LIN {X 0,Y 298.44,Z 121.432,A -85,B 0,C 180,E1 -16174.92,E2 -16174.92} C_VEL
LIN {X 0,Y 298.405,Z 121.429,A -85,B 0,C 180,E1 -16177.862,E2 -16177.862} C_VEL
LIN {X 0,Y 298.509,Z 121.421,A -85,B 0,C 180,E1 -16180.754,E2 -16180.754} C_VEL
LIN {X 0,Y 298.587,Z 121.413,A -85,B 0,C 180,E1 -16184.994,E2 -16184.994} C_VEL
LIN {X 0,Y 298.592,Z 121.415,A -85,B 0,C 180,E1 -16189.146,E2 -16189.146} C_VEL
LIN {X 0,Y 298.702,Z 121.391,A -85,B 0,C 180,E1 -16191.884,E2 -16191.884} C_VEL
LIN {X 0,Y 298.641,Z 121.406,A -85,B 0,C 180,E1 -16194.598,E2 -16194.598} C_VEL
LIN {X 0,Y 298.921,Z 121.375,A -85,B 0,C 180,E1 -16198.653,E2 -16198.653} C_VEL
LIN {X 0,Y 298.921,Z 121.361,A -85,B 0,C 180,E1 -16201.347,E2 -16201.347} C_VEL
LIN {X 0,Y 298.637,Z 121.402,A -85,B 0,C 180,E1 -16205.401,E2 -16205.401} C_VEL
LIN {X 0,Y 298.708,Z 121.401,A -85,B 0,C 180,E1 -16208.82,E2 -16208.82} C_VEL
LIN {X 0,Y 298.553,Z 121.423,A -85,B 0,C 180,E1 -16213.615,E2 -16213.615} C_VEL
LIN {X 0,Y 298.55,Z 121.407,A -85,B 0,C 180,E1 -16216.408,E2 -16216.408} C_VEL
LIN {X 0,Y 298.512,Z 121.418,A -85,B 0,C 180,E1 -16219.654,E2 -16219.654} C_VEL
LIN {X 0,Y 298.458,Z 121.428,A -85,B 0,C 180,E1 -16223.597,E2 -16223.597} C_VEL
LIN {X 0,Y 298.49,Z 121.425,A -85,B 0,C 180,E1 -16226.574,E2 -16226.574} C_VEL
LIN {X 0,Y 298.421,Z 121.432,A -85,B 0,C 180,E1 -16229.641,E2 -16229.641} C_VEL
LIN {X 0,Y 298.396,Z 121.435,A -85,B 0,C 180,E1 -16232.8,E2 -16232.8} C_VEL
LIN {X 0,Y 298.445,Z 121.436,A -85,B 0,C 180,E1 -16236.807,E2 -16236.807} C_VEL
LIN {X 0,Y 298.387,Z 121.428,A -85,B 0,C 180,E1 -16241.087,E2 -16241.087} C_VEL
LIN {X 0,Y 298.399,Z 121.435,A -85,B 0,C 180,E1 -16243.103,E2 -16243.103} C_VEL
LIN {X 0,Y 298.403,Z 121.44,A -85,B 0,C 180,E1 -16246.921,E2 -16246.921} C_VEL
LIN {X 0,Y 298.451,Z 121.59,A -85,B 0,C 180,E1 -16249.382,E2 -16249.382} C_VEL
LIN {X 0,Y 301.266,Z 131.505,A -85,B 0,C 180,E1 -16253.033,E2 -16253.033} C_VEL
LIN {X 0,Y 302.836,Z 137.275,A -85,B 0,C 180,E1 -16254.962,E2 -16254.962} C_VEL
LIN {X 0,Y 311.936,Z 155.274,A -85,B 0,C 180,E1 -16256.733,E2 -16256.733} C_VEL
LIN {X 0,Y 318.709,Z 170.292,A -85,B 0,C 180,E1 -16258.005,E2 -16258.005} C_VEL
LIN {X 0,Y 321.734,Z 187.115,A -85,B 0,C 180,E1 -16258.816,E2 -16258.816} C_VEL
LIN {X 0,Y 318.655,Z 274.997,A -85,B 0,C 180,E1 -16260.793,E2 -16260.793} C_VEL
LIN {X 0,Y 317.439,Z 289.664,A -85,B 0,C 180,E1 -16261.35,E2 -16261.35} C_VEL
LIN {X 0,Y 315.748,Z 303.63,A -85,B 0,C 180,E1 -16262.133,E2 -16262.133} C_VEL
LIN {X 0,Y 313.642,Z 317.483,A -85,B 0,C 180,E1 -16263.195,E2 -16263.195} C_VEL
LIN {X 0,Y 311.518,Z 330.032,A -85,B 0,C 180,E1 -16264.457,E2 -16264.457} C_VEL
LIN {X 0,Y 309.03,Z 342.414,A -85,B 0,C 180,E1 -16266.014,E2 -16266.014} C_VEL
LIN {X 0,Y 306.524,Z 353.602,A -85,B 0,C 180,E1 -16267.771,E2 -16267.771} C_VEL
LIN {X 0,Y 304.139,Z 363.638,A -85,B 0,C 180,E1 -16269.719,E2 -16269.719} C_VEL
LIN {X 0,Y 302.085,Z 371.989,A -85,B 0,C 180,E1 -16271.695,E2 -16271.695} C_VEL
LIN {X 0,Y 300.202,Z 379.986,A -85,B 0,C 180,E1 -16274.033,E2 -16274.033} C_VEL
LIN {X 0,Y 298.771,Z 386.446,A -85,B 0,C 180,E1 -16276.395,E2 -16276.395} C_VEL
LIN {X 0,Y 297.529,Z 392.192,A -85,B 0,C 180,E1 -16279.107,E2 -16279.107} C_VEL
LIN {X 0,Y 296.852,Z 396.392,A -85,B 0,C 180,E1 -16281.833,E2 -16281.833} C_VEL
LIN {X 0,Y 296.531,Z 399.17,A -85,B 0,C 180,E1 -16284.56,E2 -16284.56} C_VEL
LIN {X 0,Y 296.512,Z 400.597,A -85,B 0,C 180,E1 -16287.283,E2 -16287.283} C_VEL
LIN {X 0,Y 296.479,Z 400.691,A -85,B 0,C 180,E1 -16290,E2 -16290} C_VEL
LIN {X 0,Y 296.518,Z 399.447,A -85,B 0,C 180,E1 -16292.717,E2 -16292.717} C_VEL
LIN {X 0,Y 296.511,Z 396.814,A -85,B 0,C 180,E1 -16295.44,E2 -16295.44} C_VEL
LIN {X 0,Y 296.783,Z 392.722,A -85,B 0,C 180,E1 -16298.168,E2 -16298.168} C_VEL
LIN {X 0,Y 297.314,Z 387.046,A -85,B 0,C 180,E1 -16300.9,E2 -16300.9} C_VEL
LIN {X 0,Y 298.285,Z 380.643,A -85,B 0,C 180,E1 -16303.281,E2 -16303.281} C_VEL
LIN {X 0,Y 299.321,Z 373.124,A -85,B 0,C 180,E1 -16305.534,E2 -16305.534} C_VEL
LIN {X 0,Y 300.776,Z 364.3,A -85,B 0,C 180,E1 -16307.683,E2 -16307.683} C_VEL
LIN {X 0,Y 302.455,Z 354.225,A -85,B 0,C 180,E1 -16309.69,E2 -16309.69} C_VEL
LIN {X 0,Y 304.398,Z 343.006,A -85,B 0,C 180,E1 -16311.501,E2 -16311.501} C_VEL
LIN {X 0,Y 306.181,Z 331.827,A -85,B 0,C 180,E1 -16312.968,E2 -16312.968} C_VEL
LIN {X 0,Y 307.925,Z 319.653,A -85,B 0,C 180,E1 -16314.256,E2 -16314.256} C_VEL
LIN {X 0,Y 309.491,Z 306.12,A -85,B 0,C 180,E1 -16315.38,E2 -16315.38} C_VEL
LIN {X 0,Y 310.912,Z 291.992,A -85,B 0,C 180,E1 -16316.244,E2 -16316.244} C_VEL
LIN {X 0,Y 311.897,Z 278.189,A -85,B 0,C 180,E1 -16316.831,E2 -16316.831} C_VEL
LIN {X 0,Y 312.684,Z 257.755,A -85,B 0,C 180,E1 -16317.346,E2 -16317.346} C_VEL
LIN {X 0,Y 314.615,Z 183.423,A -85,B 0,C 180,E1 -16319.027,E2 -16319.027} C_VEL
LIN {X 0,Y 310.494,Z 157.724,A -85,B 0,C 180,E1 -16320.059,E2 -16320.059} C_VEL
LIN {X 0,Y 302.188,Z 137.332,A -85,B 0,C 180,E1 -16321.449,E2 -16321.449} C_VEL
LIN {X 0,Y 299.625,Z 126.323,A -85,B 0,C 180,E1 -16324.819,E2 -16324.819} C_VEL
LIN {X 0,Y 298.467,Z 121.436,A -85,B 0,C 180,E1 -16326.436,E2 -16326.436} C_VEL
LIN {X 0,Y 298.408,Z 121.44,A -85,B 0,C 180,E1 -16329.486,E2 -16329.486} C_VEL
LIN {X 0,Y 298.425,Z 121.436,A -85,B 0,C 180,E1 -16333.109,E2 -16333.109} C_VEL
LIN {X 0,Y 298.466,Z 121.429,A -85,B 0,C 180,E1 -16336.932,E2 -16336.932} C_VEL
LIN {X 0,Y 298.428,Z 121.425,A -85,B 0,C 180,E1 -16341,E2 -16341} C_VEL
LIN {X 0,Y 298.43,Z 121.436,A -85,B 0,C 180,E1 -16343.932,E2 -16343.932} C_VEL
LIN {X 0,Y 298.394,Z 121.439,A -85,B 0,C 180,E1 -16347.983,E2 -16347.983} C_VEL
LIN {X 0,Y 298.468,Z 121.429,A -85,B 0,C 180,E1 -16351.905,E2 -16351.905} C_VEL
LIN {X 0,Y 298.485,Z 121.428,A -85,B 0,C 180,E1 -16354.924,E2 -16354.924} C_VEL
LIN {X 0,Y 298.449,Z 121.432,A -85,B 0,C 180,E1 -16359.315,E2 -16359.315} C_VEL
LIN {X 0,Y 298.537,Z 121.417,A -85,B 0,C 180,E1 -16362.179,E2 -16362.179} C_VEL
LIN {X 0,Y 298.592,Z 121.416,A -85,B 0,C 180,E1 -16364.995,E2 -16364.995} C_VEL
LIN {X 0,Y 298.592,Z 121.414,A -85,B 0,C 180,E1 -16369.147,E2 -16369.147} C_VEL
LIN {X 0,Y 298.744,Z 121.395,A -85,B 0,C 180,E1 -16371.886,E2 -16371.886} C_VEL
LIN {X 0,Y 298.655,Z 121.403,A -85,B 0,C 180,E1 -16374.599,E2 -16374.599} C_VEL
LIN {X 0,Y 298.921,Z 121.374,A -85,B 0,C 180,E1 -16378.653,E2 -16378.653} C_VEL
LIN {X 0,Y 298.921,Z 121.366,A -85,B 0,C 180,E1 -16381.347,E2 -16381.347} C_VEL
LIN {X 0,Y 298.644,Z 121.407,A -85,B 0,C 180,E1 -16385.402,E2 -16385.402} C_VEL
LIN {X 0,Y 298.712,Z 121.398,A -85,B 0,C 180,E1 -16388.116,E2 -16388.116} C_VEL
LIN {X 0,Y 298.553,Z 121.42,A -85,B 0,C 180,E1 -16392.232,E2 -16392.232} C_VEL
LIN {X 0,Y 298.605,Z 121.412,A -85,B 0,C 180,E1 -16395.209,E2 -16395.209} C_VEL
LIN {X 0,Y 298.539,Z 121.417,A -85,B 0,C 180,E1 -16399.243,E2 -16399.243} C_VEL
LIN {X 0,Y 298.457,Z 121.429,A -85,B 0,C 180,E1 -16403.598,E2 -16403.598} C_VEL
LIN {X 0,Y 298.486,Z 121.424,A -85,B 0,C 180,E1 -16406.575,E2 -16406.575} C_VEL
LIN {X 0,Y 298.416,Z 121.436,A -85,B 0,C 180,E1 -16409.642,E2 -16409.642} C_VEL
LIN {X 0,Y 298.395,Z 121.436,A -85,B 0,C 180,E1 -16412.801,E2 -16412.801} C_VEL
LIN {X 0,Y 298.444,Z 121.431,A -85,B 0,C 180,E1 -16416.807,E2 -16416.807} C_VEL
LIN {X 0,Y 298.388,Z 121.439,A -85,B 0,C 180,E1 -16421.088,E2 -16421.088} C_VEL
LIN {X 0,Y 298.389,Z 121.439,A -85,B 0,C 180,E1 -16425.042,E2 -16425.042} C_VEL
LIN {X 0,Y 298.388,Z 121.439,A -85,B 0,C 180,E1 -16428.913,E2 -16428.913} C_VEL
LIN {X 0,Y 298.445,Z 121.435,A -85,B 0,C 180,E1 -16433.194,E2 -16433.194} C_VEL
LIN {X 0,Y 298.394,Z 121.44,A -85,B 0,C 180,E1 -16437.2,E2 -16437.2} C_VEL
LIN {X 0,Y 298.404,Z 121.44,A -85,B 0,C 180,E1 -16440.625,E2 -16440.625} C_VEL
LIN {X 0,Y 298.436,Z 121.472,A -85,B 0,C 180,E1 -16442.873,E2 -16442.873} C_VEL
LIN {X 0,Y 299.591,Z 126.094,A -85,B 0,C 180,E1 -16444.382,E2 -16444.382} C_VEL
LIN {X 0,Y 308.871,Z 146.99,A -85,B 0,C 180,E1 -16445.883,E2 -16445.883} C_VEL
LIN {X 0,Y 314.918,Z 162.698,A -85,B 0,C 180,E1 -16446.857,E2 -16446.857} C_VEL
LIN {X 0,Y 315.167,Z 165.643,A -85,B 0,C 180,E1 -16446.953,E2 -16446.953} C_VEL
LIN {X 0,Y 312.39,Z 262.581,A -85,B 0,C 180,E1 -16449.161,E2 -16449.161} C_VEL
LIN {X 0,Y 311.659,Z 276.3,A -85,B 0,C 180,E1 -16449.714,E2 -16449.714} C_VEL
LIN {X 0,Y 310.527,Z 289.807,A -85,B 0,C 180,E1 -16450.499,E2 -16450.499} C_VEL
LIN {X 0,Y 309.152,Z 302.098,A -85,B 0,C 180,E1 -16451.442,E2 -16451.442} C_VEL
LIN {X 0,Y 307.636,Z 313.548,A -85,B 0,C 180,E1 -16452.552,E2 -16452.552} C_VEL
LIN {X 0,Y 305.934,Z 325.457,A -85,B 0,C 180,E1 -16453.998,E2 -16453.998} C_VEL
LIN {X 0,Y 304.144,Z 336.336,A -85,B 0,C 180,E1 -16455.617,E2 -16455.617} C_VEL
LIN {X 0,Y 302.338,Z 346.911,A -85,B 0,C 180,E1 -16457.55,E2 -16457.55} C_VEL
LIN {X 0,Y 300.8,Z 355.936,A -85,B 0,C 180,E1 -16459.568,E2 -16459.568} C_VEL
LIN {X 0,Y 299.495,Z 363.328,A -85,B 0,C 180,E1 -16461.567,E2 -16461.567} C_VEL
LIN {X 0,Y 298.331,Z 370.395,A -85,B 0,C 180,E1 -16463.915,E2 -16463.915} C_VEL
LIN {X 0,Y 297.515,Z 375.339,A -85,B 0,C 180,E1 -16465.936,E2 -16465.936} C_VEL
LIN {X 0,Y 296.911,Z 380.438,A -85,B 0,C 180,E1 -16468.644,E2 -16468.644} C_VEL
LIN {X 0,Y 296.563,Z 384.053,A -85,B 0,C 180,E1 -16471.358,E2 -16471.358} C_VEL
LIN {X 0,Y 296.519,Z 386.28,A -85,B 0,C 180,E1 -16474.078,E2 -16474.078} C_VEL
LIN {X 0,Y 296.502,Z 387.182,A -85,B 0,C 180,E1 -16476.807,E2 -16476.807} C_VEL
LIN {X 0,Y 296.471,Z 386.764,A -85,B 0,C 180,E1 -16479.552,E2 -16479.552} C_VEL
LIN {X 0,Y 296.862,Z 385.003,A -85,B 0,C 180,E1 -16482.302,E2 -16482.302} C_VEL
LIN {X 0,Y 297.563,Z 381.854,A -85,B 0,C 180,E1 -16485.059,E2 -16485.059} C_VEL
LIN {X 0,Y 298.555,Z 377.171,A -85,B 0,C 180,E1 -16487.82,E2 -16487.82} C_VEL
LIN {X 0,Y 300.087,Z 371.034,A -85,B 0,C 180,E1 -16490.479,E2 -16490.479} C_VEL
LIN {X 0,Y 301.9,Z 363.692,A -85,B 0,C 180,E1 -16492.95,E2 -16492.95} C_VEL
LIN {X 0,Y 304.088,Z 355.073,A -85,B 0,C 180,E1 -16495.254,E2 -16495.254} C_VEL
LIN {X 0,Y 306.353,Z 345.552,A -85,B 0,C 180,E1 -16497.311,E2 -16497.311} C_VEL
LIN {X 0,Y 308.651,Z 335.233,A -85,B 0,C 180,E1 -16499.125,E2 -16499.125} C_VEL
LIN {X 0,Y 311.156,Z 323.794,A -85,B 0,C 180,E1 -16500.736,E2 -16500.736} C_VEL
LIN {X 0,Y 313.123,Z 312.72,A -85,B 0,C 180,E1 -16502.023,E2 -16502.023} C_VEL
LIN {X 0,Y 315.343,Z 299.818,A -85,B 0,C 180,E1 -16503.19,E2 -16503.19} C_VEL
LIN {X 0,Y 316.836,Z 287.775,A -85,B 0,C 180,E1 -16504.062,E2 -16504.062} C_VEL
LIN {X 0,Y 318.183,Z 273.727,A -85,B 0,C 180,E1 -16504.809,E2 -16504.809} C_VEL
LIN {X 0,Y 319.144,Z 259.623,A -85,B 0,C 180,E1 -16505.297,E2 -16505.297} C_VEL
LIN {X 0,Y 322.223,Z 171.012,A -85,B 0,C 180,E1 -16507.278,E2 -16507.278} C_VEL
LIN {X 0,Y 314.561,Z 154.009,A -85,B 0,C 180,E1 -16508.687,E2 -16508.687} C_VEL
LIN {X 0,Y 308.153,Z 141.521,A -85,B 0,C 180,E1 -16509.891,E2 -16509.891} C_VEL
LIN {X 0,Y 305.295,Z 136.304,A -85,B 0,C 180,E1 -16510.441,E2 -16510.441} C_VEL
LIN {X 0,Y 303.417,Z 133.303,A -85,B 0,C 180,E1 -16510.813,E2 -16510.813} C_VEL
LIN {X 0,Y 300.871,Z 131.097,A -85,B 0,C 180,E1 -16511.261,E2 -16511.261} C_VEL
LIN {X 0,Y 292.931,Z 126.669,A -85,B 0,C 180,E1 -16512.655,E2 -16512.655} C_VEL
LIN {X 0,Y 292.253,Z 125.838,A -85,B 0,C 180,E1 -16512.971,E2 -16512.971} C_VEL
LIN {X 0,Y 291.325,Z 122.315,A -85,B 0,C 180,E1 -16514.471,E2 -16514.471} C_VEL
LIN {X 0,Y 291.296,Z 122.321,A -85,B 0,C 180,E1 -16518.411,E2 -16518.411} C_VEL
LIN {X 0,Y 291.387,Z 122.315,A -85,B 0,C 180,E1 -16522.916,E2 -16522.916} C_VEL
LIN {X 0,Y 291.345,Z 122.316,A -85,B 0,C 180,E1 -16526.301,E2 -16526.301} C_VEL
LIN {X 0,Y 291.366,Z 122.308,A -85,B 0,C 180,E1 -16530.268,E2 -16530.268} C_VEL
LIN {X 0,Y 291.36,Z 122.309,A -85,B 0,C 180,E1 -16534.266,E2 -16534.266} C_VEL
LIN {X 0,Y 291.366,Z 122.306,A -85,B 0,C 180,E1 -16537.298,E2 -16537.298} C_VEL
LIN {X 0,Y 291.46,Z 122.305,A -85,B 0,C 180,E1 -16540.27,E2 -16540.27} C_VEL
LIN {X 0,Y 291.499,Z 122.298,A -85,B 0,C 180,E1 -16544.665,E2 -16544.665} C_VEL
LIN {X 0,Y 291.536,Z 122.295,A -85,B 0,C 180,E1 -16548.88,E2 -16548.88} C_VEL
LIN {X 0,Y 291.655,Z 122.267,A -85,B 0,C 180,E1 -16551.687,E2 -16551.687} C_VEL
LIN {X 0,Y 291.61,Z 122.283,A -85,B 0,C 180,E1 -16554.468,E2 -16554.468} C_VEL
LIN {X 0,Y 291.887,Z 122.251,A -85,B 0,C 180,E1 -16558.62,E2 -16558.62} C_VEL
LIN {X 0,Y 291.887,Z 122.237,A -85,B 0,C 180,E1 -16561.379,E2 -16561.379} C_VEL
LIN {X 0,Y 291.606,Z 122.276,A -85,B 0,C 180,E1 -16565.532,E2 -16565.532} C_VEL
LIN {X 0,Y 291.668,Z 122.278,A -85,B 0,C 180,E1 -16568.91,E2 -16568.91} C_VEL
LIN {X 0,Y 291.519,Z 122.291,A -85,B 0,C 180,E1 -16572.531,E2 -16572.531} C_VEL
LIN {X 0,Y 291.556,Z 122.282,A -85,B 0,C 180,E1 -16575.376,E2 -16575.376} C_VEL
LIN {X 0,Y 291.452,Z 122.297,A -85,B 0,C 180,E1 -16579.875,E2 -16579.875} C_VEL
LIN {X 0,Y 291.401,Z 122.304,A -85,B 0,C 180,E1 -16584.205,E2 -16584.205} C_VEL
LIN {X 0,Y 291.423,Z 122.307,A -85,B 0,C 180,E1 -16587.271,E2 -16587.271} C_VEL
LIN {X 0,Y 291.338,Z 122.318,A -85,B 0,C 180,E1 -16590.437,E2 -16590.437} C_VEL
LIN {X 0,Y 291.345,Z 122.319,A -85,B 0,C 180,E1 -16593.698,E2 -16593.698} C_VEL
LIN {X 0,Y 291.373,Z 122.316,A -85,B 0,C 180,E1 -16597.253,E2 -16597.253} C_VEL
LIN {X 0,Y 291.332,Z 122.3,A -85,B 0,C 180,E1 -16600.642,E2 -16600.642} C_VEL
LIN {X 0,Y 291.29,Z 122.308,A -85,B 0,C 180,E1 -16604.402,E2 -16604.402} C_VEL
LIN {X 0,Y 291.367,Z 122.352,A -85,B 0,C 180,E1 -16608.395,E2 -16608.395} C_VEL
LIN {X 0,Y 294.066,Z 131.907,A -85,B 0,C 180,E1 -16612.062,E2 -16612.062} C_VEL
LIN {X 0,Y 295.437,Z 136.791,A -85,B 0,C 180,E1 -16613.836,E2 -16613.836} C_VEL
LIN {X 0,Y 303.07,Z 151.502,A -85,B 0,C 180,E1 -16615.411,E2 -16615.411} C_VEL
LIN {X 0,Y 311.133,Z 168.352,A -85,B 0,C 180,E1 -16616.991,E2 -16616.991} C_VEL
LIN {X 0,Y 313.243,Z 173.632,A -85,B 0,C 180,E1 -16617.41,E2 -16617.41} C_VEL
LIN {X 0,Y 315.791,Z 188.416,A -85,B 0,C 180,E1 -16618.133,E2 -16618.133} C_VEL
LIN {X 0,Y 312.601,Z 275.339,A -85,B 0,C 180,E1 -16620.124,E2 -16620.124} C_VEL
LIN {X 0,Y 311.345,Z 289.824,A -85,B 0,C 180,E1 -16620.689,E2 -16620.689} C_VEL
LIN {X 0,Y 309.516,Z 304.269,A -85,B 0,C 180,E1 -16621.521,E2 -16621.521} C_VEL
LIN {X 0,Y 307.347,Z 317.946,A -85,B 0,C 180,E1 -16622.6,E2 -16622.6} C_VEL
LIN {X 0,Y 305.174,Z 330.231,A -85,B 0,C 180,E1 -16623.868,E2 -16623.868} C_VEL
LIN {X 0,Y 302.569,Z 342.657,A -85,B 0,C 180,E1 -16625.468,E2 -16625.468} C_VEL
LIN {X 0,Y 299.964,Z 353.753,A -85,B 0,C 180,E1 -16627.258,E2 -16627.258} C_VEL
LIN {X 0,Y 297.459,Z 363.736,A -85,B 0,C 180,E1 -16629.243,E2 -16629.243} C_VEL
LIN {X 0,Y 295.002,Z 373.271,A -85,B 0,C 180,E1 -16631.599,E2 -16631.599} C_VEL
LIN {X 0,Y 293.363,Z 379.811,A -85,B 0,C 180,E1 -16633.584,E2 -16633.584} C_VEL
LIN {X 0,Y 291.848,Z 386.424,A -85,B 0,C 180,E1 -16636.065,E2 -16636.065} C_VEL
LIN {X 0,Y 290.524,Z 392.137,A -85,B 0,C 180,E1 -16638.841,E2 -16638.841} C_VEL
LIN {X 0,Y 289.809,Z 396.306,A -85,B 0,C 180,E1 -16641.633,E2 -16641.633} C_VEL
LIN {X 0,Y 289.426,Z 399.204,A -85,B 0,C 180,E1 -16644.614,E2 -16644.614} C_VEL
LIN {X 0,Y 289.416,Z 400.454,A -85,B 0,C 180,E1 -16647.216,E2 -16647.216} C_VEL
LIN {X 0,Y 289.398,Z 400.52,A -85,B 0,C 180,E1 -16650,E2 -16650} C_VEL
LIN {X 0,Y 289.421,Z 399.241,A -85,B 0,C 180,E1 -16652.783,E2 -16652.783} C_VEL
LIN {X 0,Y 289.434,Z 396.574,A -85,B 0,C 180,E1 -16655.574,E2 -16655.574} C_VEL
LIN {X 0,Y 289.718,Z 392.45,A -85,B 0,C 180,E1 -16658.369,E2 -16658.369} C_VEL
LIN {X 0,Y 290.122,Z 388.36,A -85,B 0,C 180,E1 -16660.467,E2 -16660.467} C_VEL
LIN {X 0,Y 290.841,Z 383.247,A -85,B 0,C 180,E1 -16662.561,E2 -16662.561} C_VEL
LIN {X 0,Y 292.008,Z 375.941,A -85,B 0,C 180,E1 -16664.994,E2 -16664.994} C_VEL
LIN {X 0,Y 293.136,Z 368.263,A -85,B 0,C 180,E1 -16667.079,E2 -16667.079} C_VEL
LIN {X 0,Y 294.815,Z 359.054,A -85,B 0,C 180,E1 -16669.134,E2 -16669.134} C_VEL
LIN {X 0,Y 296.386,Z 349.857,A -85,B 0,C 180,E1 -16670.835,E2 -16670.835} C_VEL
LIN {X 0,Y 298.382,Z 338.889,A -85,B 0,C 180,E1 -16672.504,E2 -16672.504} C_VEL
LIN {X 0,Y 300.217,Z 326.747,A -85,B 0,C 180,E1 -16674.013,E2 -16674.013} C_VEL
LIN {X 0,Y 301.87,Z 315.299,A -85,B 0,C 180,E1 -16675.143,E2 -16675.143} C_VEL
LIN {X 0,Y 303.311,Z 302.88,A -85,B 0,C 180,E1 -16676.119,E2 -16676.119} C_VEL
LIN {X 0,Y 304.703,Z 288.433,A -85,B 0,C 180,E1 -16676.96,E2 -16676.96} C_VEL
LIN {X 0,Y 305.701,Z 273.863,A -85,B 0,C 180,E1 -16677.513,E2 -16677.513} C_VEL
LIN {X 0,Y 308.253,Z 184.312,A -85,B 0,C 180,E1 -16679.592,E2 -16679.592} C_VEL
LIN {X 0,Y 304.502,Z 160.641,A -85,B 0,C 180,E1 -16680.568,E2 -16680.568} C_VEL
LIN {X 0,Y 297.951,Z 144.295,A -85,B 0,C 180,E1 -16681.677,E2 -16681.677} C_VEL
LIN {X 0,Y 294.952,Z 137.255,A -85,B 0,C 180,E1 -16682.196,E2 -16682.196} C_VEL
LIN {X 0,Y 292.386,Z 126.362,A -85,B 0,C 180,E1 -16685.653,E2 -16685.653} C_VEL
LIN {X 0,Y 291.428,Z 122.313,A -85,B 0,C 180,E1 -16687.023,E2 -16687.023} C_VEL
LIN {X 0,Y 291.334,Z 122.319,A -85,B 0,C 180,E1 -16690.642,E2 -16690.642} C_VEL
LIN {X 0,Y 291.341,Z 122.318,A -85,B 0,C 180,E1 -16694.392,E2 -16694.392} C_VEL
LIN {X 0,Y 291.386,Z 122.312,A -85,B 0,C 180,E1 -16698.391,E2 -16698.391} C_VEL
LIN {X 0,Y 291.376,Z 122.301,A -85,B 0,C 180,E1 -16701.162,E2 -16701.162} C_VEL
LIN {X 0,Y 291.384,Z 122.312,A -85,B 0,C 180,E1 -16704.629,E2 -16704.629} C_VEL
LIN {X 0,Y 291.371,Z 122.315,A -85,B 0,C 180,E1 -16707.951,E2 -16707.951} C_VEL
LIN {X 0,Y 291.384,Z 122.311,A -85,B 0,C 180,E1 -16711.159,E2 -16711.159} C_VEL
LIN {X 0,Y 291.419,Z 122.307,A -85,B 0,C 180,E1 -16714.272,E2 -16714.272} C_VEL
LIN {X 0,Y 291.38,Z 122.315,A -85,B 0,C 180,E1 -16717.3,E2 -16717.3} C_VEL
LIN {X 0,Y 291.457,Z 122.301,A -85,B 0,C 180,E1 -16720.27,E2 -16720.27} C_VEL
LIN {X 0,Y 291.554,Z 122.294,A -85,B 0,C 180,E1 -16724.624,E2 -16724.624} C_VEL
LIN {X 0,Y 291.535,Z 122.293,A -85,B 0,C 180,E1 -16728.881,E2 -16728.881} C_VEL
LIN {X 0,Y 291.696,Z 122.273,A -85,B 0,C 180,E1 -16731.688,E2 -16731.688} C_VEL
LIN {X 0,Y 291.626,Z 122.277,A -85,B 0,C 180,E1 -16734.468,E2 -16734.468} C_VEL
LIN {X 0,Y 291.887,Z 122.251,A -85,B 0,C 180,E1 -16738.621,E2 -16738.621} C_VEL
LIN {X 0,Y 291.887,Z 122.241,A -85,B 0,C 180,E1 -16741.38,E2 -16741.38} C_VEL
LIN {X 0,Y 291.659,Z 122.275,A -85,B 0,C 180,E1 -16746.552,E2 -16746.552} C_VEL
LIN {X 0,Y 291.571,Z 122.282,A -85,B 0,C 180,E1 -16749.714,E2 -16749.714} C_VEL
LIN {X 0,Y 291.521,Z 122.298,A -85,B 0,C 180,E1 -16753.951,E2 -16753.951} C_VEL
LIN {X 0,Y 291.486,Z 122.293,A -85,B 0,C 180,E1 -16756.818,E2 -16756.818} C_VEL
LIN {X 0,Y 291.45,Z 122.305,A -85,B 0,C 180,E1 -16759.875,E2 -16759.875} C_VEL
LIN {X 0,Y 291.4,Z 122.303,A -85,B 0,C 180,E1 -16764.206,E2 -16764.206} C_VEL
LIN {X 0,Y 291.42,Z 122.308,A -85,B 0,C 180,E1 -16767.272,E2 -16767.272} C_VEL
LIN {X 0,Y 291.334,Z 122.315,A -85,B 0,C 180,E1 -16770.438,E2 -16770.438} C_VEL
LIN {X 0,Y 291.344,Z 122.318,A -85,B 0,C 180,E1 -16773.699,E2 -16773.699} C_VEL
LIN {X 0,Y 291.372,Z 122.311,A -85,B 0,C 180,E1 -16777.253,E2 -16777.253} C_VEL
LIN {X 0,Y 291.333,Z 122.321,A -85,B 0,C 180,E1 -16780.643,E2 -16780.643} C_VEL
LIN {X 0,Y 291.315,Z 122.323,A -85,B 0,C 180,E1 -16784.398,E2 -16784.398} C_VEL
LIN {X 0,Y 291.328,Z 122.322,A -85,B 0,C 180,E1 -16788.405,E2 -16788.405} C_VEL
LIN {X 0,Y 291.348,Z 122.305,A -85,B 0,C 180,E1 -16791.158,E2 -16791.158} C_VEL
LIN {X 0,Y 291.362,Z 122.318,A -85,B 0,C 180,E1 -16794.627,E2 -16794.627} C_VEL
LIN {X 0,Y 291.367,Z 122.316,A -85,B 0,C 180,E1 -16797.95,E2 -16797.95} C_VEL
LIN {X 0,Y 291.39,Z 122.313,A -85,B 0,C 180,E1 -16802.141,E2 -16802.141} C_VEL
LIN {X 0,Y 291.397,Z 122.542,A -85,B 0,C 180,E1 -16802.337,E2 -16802.337} C_VEL
LIN {X 0,Y 292.364,Z 126.299,A -85,B 0,C 180,E1 -16803.591,E2 -16803.591} C_VEL
LIN {X 0,Y 300.522,Z 144.106,A -85,B 0,C 180,E1 -16804.964,E2 -16804.964} C_VEL
LIN {X 0,Y 307.832,Z 162.323,A -85,B 0,C 180,E1 -16806.178,E2 -16806.178} C_VEL
LIN {X 0,Y 308.799,Z 165.052,A -85,B 0,C 180,E1 -16806.341,E2 -16806.341} C_VEL
LIN {X 0,Y 305.952,Z 262.733,A -85,B 0,C 180,E1 -16808.613,E2 -16808.613} C_VEL
LIN {X 0,Y 305.187,Z 276.458,A -85,B 0,C 180,E1 -16809.176,E2 -16809.176} C_VEL
LIN {X 0,Y 304.024,Z 289.966,A -85,B 0,C 180,E1 -16809.976,E2 -16809.976} C_VEL
LIN {X 0,Y 302.483,Z 303.136,A -85,B 0,C 180,E1 -16811.018,E2 -16811.018} C_VEL
LIN {X 0,Y 300.93,Z 314.417,A -85,B 0,C 180,E1 -16812.15,E2 -16812.15} C_VEL
LIN {X 0,Y 299.145,Z 326.205,A -85,B 0,C 180,E1 -16813.625,E2 -16813.625} C_VEL
LIN {X 0,Y 297.312,Z 336.984,A -85,B 0,C 180,E1 -16815.279,E2 -16815.279} C_VEL
LIN {X 0,Y 295.509,Z 347.152,A -85,B 0,C 180,E1 -16817.187,E2 -16817.187} C_VEL
LIN {X 0,Y 293.859,Z 356.435,A -85,B 0,C 180,E1 -16819.319,E2 -16819.319} C_VEL
LIN {X 0,Y 292.497,Z 363.769,A -85,B 0,C 180,E1 -16821.363,E2 -16821.363} C_VEL
LIN {X 0,Y 291.279,Z 370.784,A -85,B 0,C 180,E1 -16823.767,E2 -16823.767} C_VEL
LIN {X 0,Y 290.443,Z 375.68,A -85,B 0,C 180,E1 -16825.837,E2 -16825.837} C_VEL
LIN {X 0,Y 290.013,Z 379.632,A -85,B 0,C 180,E1 -16827.917,E2 -16827.917} C_VEL
LIN {X 0,Y 289.6,Z 382.699,A -85,B 0,C 180,E1 -16830,E2 -16830} C_VEL
LIN {X 0,Y 289.481,Z 385.567,A -85,B 0,C 180,E1 -16832.783,E2 -16832.783} C_VEL
LIN {X 0,Y 289.434,Z 387.089,A -85,B 0,C 180,E1 -16835.574,E2 -16835.574} C_VEL
LIN {X 0,Y 289.337,Z 387.294,A -85,B 0,C 180,E1 -16838.38,E2 -16838.38} C_VEL
LIN {X 0,Y 289.528,Z 386.167,A -85,B 0,C 180,E1 -16841.198,E2 -16841.198} C_VEL
LIN {X 0,Y 290.183,Z 383.678,A -85,B 0,C 180,E1 -16844.016,E2 -16844.016} C_VEL
LIN {X 0,Y 291.051,Z 379.723,A -85,B 0,C 180,E1 -16846.844,E2 -16846.844} C_VEL
LIN {X 0,Y 292.469,Z 374.17,A -85,B 0,C 180,E1 -16849.659,E2 -16849.659} C_VEL
LIN {X 0,Y 294.109,Z 367.864,A -85,B 0,C 180,E1 -16852.109,E2 -16852.109} C_VEL
LIN {X 0,Y 296.215,Z 359.98,A -85,B 0,C 180,E1 -16854.532,E2 -16854.532} C_VEL
LIN {X 0,Y 298.363,Z 351.709,A -85,B 0,C 180,E1 -16856.587,E2 -16856.587} C_VEL
LIN {X 0,Y 300.755,Z 341.702,A -85,B 0,C 180,E1 -16858.623,E2 -16858.623} C_VEL
LIN {X 0,Y 303.124,Z 331.626,A -85,B 0,C 180,E1 -16860.284,E2 -16860.284} C_VEL
LIN {X 0,Y 305.711,Z 319.404,A -85,B 0,C 180,E1 -16861.921,E2 -16861.921} C_VEL
LIN {X 0,Y 307.97,Z 307.274,A -85,B 0,C 180,E1 -16863.209,E2 -16863.209} C_VEL
LIN {X 0,Y 309.989,Z 293.778,A -85,B 0,C 180,E1 -16864.33,E2 -16864.33} C_VEL
LIN {X 0,Y 311.6,Z 279.631,A -85,B 0,C 180,E1 -16865.209,E2 -16865.209} C_VEL
LIN {X 0,Y 312.793,Z 265.42,A -85,B 0,C 180,E1 -16865.812,E2 -16865.812} C_VEL
LIN {X 0,Y 313.742,Z 243.274,A -85,B 0,C 180,E1 -16866.369,E2 -16866.369} C_VEL
LIN {X 0,Y 316.316,Z 173.613,A -85,B 0,C 180,E1 -16867.93,E2 -16867.93} C_VEL
LIN {X 0,Y 310.974,Z 161.025,A -85,B 0,C 180,E1 -16868.961,E2 -16868.961} C_VEL
LIN {X 0,Y 303.586,Z 146.257,A -85,B 0,C 180,E1 -16870.396,E2 -16870.396} C_VEL
LIN {X 0,Y 296.791,Z 134.136,A -85,B 0,C 180,E1 -16871.761,E2 -16871.761} C_VEL
LIN {X 0,Y 292.475,Z 126.533,A -85,B 0,C 180,E1 -16872.686,E2 -16872.686} C_VEL
LIN {X 0,Y 292.253,Z 125.838,A -85,B 0,C 180,E1 -16872.971,E2 -16872.971} C_VEL
LIN {X 0,Y 291.13,Z 124.464,A -85,B 0,C 180,E1 -16873.674,E2 -16873.674} C_VEL
LIN {X 0,Y 287.887,Z 123.379,A -85,B 0,C 180,E1 -16874.828,E2 -16874.828} C_VEL
LIN {X 0,Y 284.903,Z 123.179,A -85,B 0,C 180,E1 -16876.049,E2 -16876.049} C_VEL
LIN {X 0,Y 284.209,Z 123.196,A -85,B 0,C 180,E1 -16876.847,E2 -16876.847} C_VEL
LIN {X 0,Y 284.257,Z 123.18,A -85,B 0,C 180,E1 -16880.036,E2 -16880.036} C_VEL
LIN {X 0,Y 284.319,Z 123.189,A -85,B 0,C 180,E1 -16883.612,E2 -16883.612} C_VEL
LIN {X 0,Y 284.307,Z 123.19,A -85,B 0,C 180,E1 -16887.19,E2 -16887.19} C_VEL
LIN {X 0,Y 284.338,Z 123.184,A -85,B 0,C 180,E1 -16890.373,E2 -16890.373} C_VEL
LIN {X 0,Y 284.306,Z 123.186,A -85,B 0,C 180,E1 -16893.579,E2 -16893.579} C_VEL
LIN {X 0,Y 284.329,Z 123.187,A -85,B 0,C 180,E1 -16896.703,E2 -16896.703} C_VEL
LIN {X 0,Y 284.378,Z 123.187,A -85,B 0,C 180,E1 -16899.904,E2 -16899.904} C_VEL
LIN {X 0,Y 284.449,Z 123.178,A -85,B 0,C 180,E1 -16904.492,E2 -16904.492} C_VEL
LIN {X 0,Y 284.488,Z 123.175,A -85,B 0,C 180,E1 -16908.601,E2 -16908.601} C_VEL
LIN {X 0,Y 284.611,Z 123.143,A -85,B 0,C 180,E1 -16911.479,E2 -16911.479} C_VEL
LIN {X 0,Y 284.579,Z 123.16,A -85,B 0,C 180,E1 -16914.331,E2 -16914.331} C_VEL
LIN {X 0,Y 284.853,Z 123.128,A -85,B 0,C 180,E1 -16918.586,E2 -16918.586} C_VEL
LIN {X 0,Y 284.853,Z 123.113,A -85,B 0,C 180,E1 -16921.414,E2 -16921.414} C_VEL
LIN {X 0,Y 284.644,Z 123.142,A -85,B 0,C 180,E1 -16927.091,E2 -16927.091} C_VEL
LIN {X 0,Y 284.515,Z 123.165,A -85,B 0,C 180,E1 -16929.957,E2 -16929.957} C_VEL
LIN {X 0,Y 284.483,Z 123.172,A -85,B 0,C 180,E1 -16934.302,E2 -16934.302} C_VEL
LIN {X 0,Y 284.426,Z 123.17,A -85,B 0,C 180,E1 -16937.248,E2 -16937.248} C_VEL
LIN {X 0,Y 284.38,Z 123.175,A -85,B 0,C 180,E1 -16940.242,E2 -16940.242} C_VEL
LIN {X 0,Y 284.37,Z 123.181,A -85,B 0,C 180,E1 -16943.875,E2 -16943.875} C_VEL
LIN {X 0,Y 284.398,Z 123.183,A -85,B 0,C 180,E1 -16947.173,E2 -16947.173} C_VEL
LIN {X 0,Y 284.296,Z 123.194,A -85,B 0,C 180,E1 -16951.274,E2 -16951.274} C_VEL
LIN {X 0,Y 284.341,Z 123.185,A -85,B 0,C 180,E1 -16955.348,E2 -16955.348} C_VEL
LIN {X 0,Y 284.309,Z 123.185,A -85,B 0,C 180,E1 -16958.169,E2 -16958.169} C_VEL
LIN {X 0,Y 284.27,Z 123.2,A -85,B 0,C 180,E1 -16962.124,E2 -16962.124} C_VEL
LIN {X 0,Y 284.256,Z 123.198,A -85,B 0,C 180,E1 -16966.189,E2 -16966.189} C_VEL
LIN {X 0,Y 284.302,Z 123.318,A -85,B 0,C 180,E1 -16967.418,E2 -16967.418} C_VEL
LIN {X 0,Y 287.035,Z 132.498,A -85,B 0,C 180,E1 -16971.116,E2 -16971.116} C_VEL
LIN {X 0,Y 288.156,Z 136.684,A -85,B 0,C 180,E1 -16972.668,E2 -16972.668} C_VEL
LIN {X 0,Y 295.869,Z 150.998,A -85,B 0,C 180,E1 -16974.336,E2 -16974.336} C_VEL
LIN {X 0,Y 303.934,Z 167.594,A -85,B 0,C 180,E1 -16975.998,E2 -16975.998} C_VEL
LIN {X 0,Y 307.666,Z 176.255,A -85,B 0,C 180,E1 -16976.754,E2 -16976.754} C_VEL
LIN {X 0,Y 309.895,Z 190,A -85,B 0,C 180,E1 -16977.431,E2 -16977.431} C_VEL
LIN {X 0,Y 306.684,Z 274.483,A -85,B 0,C 180,E1 -16979.391,E2 -16979.391} C_VEL
LIN {X 0,Y 305.375,Z 289.227,A -85,B 0,C 180,E1 -16979.963,E2 -16979.963} C_VEL
LIN {X 0,Y 303.673,Z 302.659,A -85,B 0,C 180,E1 -16980.731,E2 -16980.731} C_VEL
LIN {X 0,Y 301.421,Z 316.651,A -85,B 0,C 180,E1 -16981.826,E2 -16981.826} C_VEL
LIN {X 0,Y 299.09,Z 329.156,A -85,B 0,C 180,E1 -16983.106,E2 -16983.106} C_VEL
LIN {X 0,Y 296.8,Z 340.084,A -85,B 0,C 180,E1 -16984.504,E2 -16984.504} C_VEL
LIN {X 0,Y 294.365,Z 350.118,A -85,B 0,C 180,E1 -16986.054,E2 -16986.054} C_VEL
LIN {X 0,Y 291.665,Z 360.729,A -85,B 0,C 180,E1 -16988.069,E2 -16988.069} C_VEL
LIN {X 0,Y 289.282,Z 369.505,A -85,B 0,C 180,E1 -16990.115,E2 -16990.115} C_VEL
LIN {X 0,Y 286.979,Z 377.936,A -85,B 0,C 180,E1 -16992.542,E2 -16992.542} C_VEL
LIN {X 0,Y 285.349,Z 384.743,A -85,B 0,C 180,E1 -16995.012,E2 -16995.012} C_VEL
LIN {X 0,Y 284.095,Z 389.444,A -85,B 0,C 180,E1 -16997.135,E2 -16997.135} C_VEL
LIN {X 0,Y 283.076,Z 394.335,A -85,B 0,C 180,E1 -16999.992,E2 -16999.992} C_VEL
LIN {X 0,Y 282.498,Z 397.752,A -85,B 0,C 180,E1 -17002.854,E2 -17002.854} C_VEL
LIN {X 0,Y 282.292,Z 399.792,A -85,B 0,C 180,E1 -17005.716,E2 -17005.716} C_VEL
LIN {X 0,Y 282.311,Z 400.495,A -85,B 0,C 180,E1 -17008.573,E2 -17008.573} C_VEL
LIN {X 0,Y 282.321,Z 399.857,A -85,B 0,C 180,E1 -17011.426,E2 -17011.426} C_VEL
LIN {X 0,Y 282.327,Z 399.03,A -85,B 0,C 180,E1 -17012.853,E2 -17012.853} C_VEL
LIN {X 0,Y 282.34,Z 396.332,A -85,B 0,C 180,E1 -17015.714,E2 -17015.714} C_VEL
LIN {X 0,Y 282.648,Z 392.176,A -85,B 0,C 180,E1 -17018.58,E2 -17018.58} C_VEL
LIN {X 0,Y 283.266,Z 386.435,A -85,B 0,C 180,E1 -17021.448,E2 -17021.448} C_VEL
LIN {X 0,Y 284.339,Z 379.959,A -85,B 0,C 180,E1 -17023.945,E2 -17023.945} C_VEL
LIN {X 0,Y 285.461,Z 372.642,A -85,B 0,C 180,E1 -17026.225,E2 -17026.225} C_VEL
LIN {X 0,Y 287.162,Z 363.446,A -85,B 0,C 180,E1 -17028.551,E2 -17028.551} C_VEL
LIN {X 0,Y 288.996,Z 353.262,A -85,B 0,C 180,E1 -17030.647,E2 -17030.647} C_VEL
LIN {X 0,Y 291.126,Z 341.854,A -85,B 0,C 180,E1 -17032.534,E2 -17032.534} C_VEL
LIN {X 0,Y 293.021,Z 330.489,A -85,B 0,C 180,E1 -17034.063,E2 -17034.063} C_VEL
LIN {X 0,Y 294.919,Z 318.063,A -85,B 0,C 180,E1 -17035.4,E2 -17035.4} C_VEL
LIN {X 0,Y 296.532,Z 305.322,A -85,B 0,C 180,E1 -17036.479,E2 -17036.479} C_VEL
LIN {X 0,Y 298.049,Z 291.028,A -85,B 0,C 180,E1 -17037.375,E2 -17037.375} C_VEL
LIN {X 0,Y 299.082,Z 276.903,A -85,B 0,C 180,E1 -17037.984,E2 -17037.984} C_VEL
LIN {X 0,Y 300.032,Z 252.306,A -85,B 0,C 180,E1 -17038.602,E2 -17038.602} C_VEL
LIN {X 0,Y 301.876,Z 184.729,A -85,B 0,C 180,E1 -17040.196,E2 -17040.196} C_VEL
LIN {X 0,Y 298.369,Z 162.643,A -85,B 0,C 180,E1 -17041.139,E2 -17041.139} C_VEL
LIN {X 0,Y 290.54,Z 143.677,A -85,B 0,C 180,E1 -17042.506,E2 -17042.506} C_VEL
LIN {X 0,Y 287.692,Z 136.982,A -85,B 0,C 180,E1 -17043.046,E2 -17043.046} C_VEL
LIN {X 0,Y 285.118,Z 126.235,A -85,B 0,C 180,E1 -17046.592,E2 -17046.592} C_VEL
LIN {X 0,Y 284.337,Z 123.195,A -85,B 0,C 180,E1 -17047.679,E2 -17047.679} C_VEL
LIN {X 0,Y 284.281,Z 123.201,A -85,B 0,C 180,E1 -17051.874,E2 -17051.874} C_VEL
LIN {X 0,Y 284.317,Z 123.192,A -85,B 0,C 180,E1 -17056.201,E2 -17056.201} C_VEL
LIN {X 0,Y 284.35,Z 123.18,A -85,B 0,C 180,E1 -17060.013,E2 -17060.013} C_VEL
LIN {X 0,Y 284.35,Z 123.188,A -85,B 0,C 180,E1 -17063.617,E2 -17063.617} C_VEL
LIN {X 0,Y 284.307,Z 123.192,A -85,B 0,C 180,E1 -17067.189,E2 -17067.189} C_VEL
LIN {X 0,Y 284.358,Z 123.185,A -85,B 0,C 180,E1 -17070.376,E2 -17070.376} C_VEL
LIN {X 0,Y 284.379,Z 123.186,A -85,B 0,C 180,E1 -17073.587,E2 -17073.587} C_VEL
LIN {X 0,Y 284.365,Z 123.183,A -85,B 0,C 180,E1 -17076.707,E2 -17076.707} C_VEL
LIN {X 0,Y 284.402,Z 123.177,A -85,B 0,C 180,E1 -17081.262,E2 -17081.262} C_VEL
LIN {X 0,Y 284.491,Z 123.173,A -85,B 0,C 180,E1 -17084.459,E2 -17084.459} C_VEL
LIN {X 0,Y 284.487,Z 123.167,A -85,B 0,C 180,E1 -17088.602,E2 -17088.602} C_VEL
LIN {X 0,Y 284.648,Z 123.151,A -85,B 0,C 180,E1 -17091.481,E2 -17091.481} C_VEL
LIN {X 0,Y 284.596,Z 123.152,A -85,B 0,C 180,E1 -17094.331,E2 -17094.331} C_VEL
LIN {X 0,Y 284.853,Z 123.127,A -85,B 0,C 180,E1 -17098.586,E2 -17098.586} C_VEL
LIN {X 0,Y 284.853,Z 123.117,A -85,B 0,C 180,E1 -17101.414,E2 -17101.414} C_VEL
LIN {X 0,Y 284.653,Z 123.149,A -85,B 0,C 180,E1 -17107.091,E2 -17107.091} C_VEL
LIN {X 0,Y 284.517,Z 123.159,A -85,B 0,C 180,E1 -17109.957,E2 -17109.957} C_VEL
LIN {X 0,Y 284.481,Z 123.173,A -85,B 0,C 180,E1 -17114.303,E2 -17114.303} C_VEL
LIN {X 0,Y 284.425,Z 123.173,A -85,B 0,C 180,E1 -17117.249,E2 -17117.249} C_VEL
LIN {X 0,Y 284.38,Z 123.185,A -85,B 0,C 180,E1 -17120.242,E2 -17120.242} C_VEL
LIN {X 0,Y 284.369,Z 123.18,A -85,B 0,C 180,E1 -17123.876,E2 -17123.876} C_VEL
LIN {X 0,Y 284.395,Z 123.182,A -85,B 0,C 180,E1 -17127.173,E2 -17127.173} C_VEL
LIN {X 0,Y 284.293,Z 123.191,A -85,B 0,C 180,E1 -17131.275,E2 -17131.275} C_VEL
LIN {X 0,Y 284.341,Z 123.19,A -85,B 0,C 180,E1 -17135.348,E2 -17135.348} C_VEL
LIN {X 0,Y 284.308,Z 123.191,A -85,B 0,C 180,E1 -17138.17,E2 -17138.17} C_VEL
LIN {X 0,Y 284.269,Z 123.194,A -85,B 0,C 180,E1 -17142.125,E2 -17142.125} C_VEL
LIN {X 0,Y 284.269,Z 123.195,A -85,B 0,C 180,E1 -17146.192,E2 -17146.192} C_VEL
LIN {X 0,Y 284.307,Z 123.187,A -85,B 0,C 180,E1 -17150.024,E2 -17150.024} C_VEL
LIN {X 0,Y 284.331,Z 123.193,A -85,B 0,C 180,E1 -17153.614,E2 -17153.614} C_VEL
LIN {X 0,Y 284.307,Z 123.195,A -85,B 0,C 180,E1 -17157.191,E2 -17157.191} C_VEL
LIN {X 0,Y 284.34,Z 123.218,A -85,B 0,C 180,E1 -17161.639,E2 -17161.639} C_VEL
LIN {X 0,Y 285.099,Z 126.354,A -85,B 0,C 180,E1 -17162.744,E2 -17162.744} C_VEL
LIN {X 0,Y 293.079,Z 143.35,A -85,B 0,C 180,E1 -17164.143,E2 -17164.143} C_VEL
LIN {X 0,Y 300.243,Z 160.773,A -85,B 0,C 180,E1 -17165.38,E2 -17165.38} C_VEL
LIN {X 0,Y 302.447,Z 166.736,A -85,B 0,C 180,E1 -17165.762,E2 -17165.762} C_VEL
LIN {X 0,Y 299.542,Z 262.872,A -85,B 0,C 180,E1 -17168.042,E2 -17168.042} C_VEL
LIN {X 0,Y 298.737,Z 276.607,A -85,B 0,C 180,E1 -17168.614,E2 -17168.614} C_VEL
LIN {X 0,Y 297.538,Z 290.117,A -85,B 0,C 180,E1 -17169.43,E2 -17169.43} C_VEL
LIN {X 0,Y 296.066,Z 302.413,A -85,B 0,C 180,E1 -17170.41,E2 -17170.41} C_VEL
LIN {X 0,Y 294.237,Z 315.278,A -85,B 0,C 180,E1 -17171.73,E2 -17171.73} C_VEL
LIN {X 0,Y 292.374,Z 326.945,A -85,B 0,C 180,E1 -17173.235,E2 -17173.235} C_VEL
LIN {X 0,Y 290.498,Z 337.627,A -85,B 0,C 180,E1 -17174.926,E2 -17174.926} C_VEL
LIN {X 0,Y 288.82,Z 346.593,A -85,B 0,C 180,E1 -17176.635,E2 -17176.635} C_VEL
LIN {X 0,Y 287.165,Z 355.591,A -85,B 0,C 180,E1 -17178.709,E2 -17178.709} C_VEL
LIN {X 0,Y 285.506,Z 364.209,A -85,B 0,C 180,E1 -17181.15,E2 -17181.15} C_VEL
LIN {X 0,Y 284.231,Z 371.173,A -85,B 0,C 180,E1 -17183.612,E2 -17183.612} C_VEL
LIN {X 0,Y 283.373,Z 376.021,A -85,B 0,C 180,E1 -17185.733,E2 -17185.733} C_VEL
LIN {X 0,Y 282.921,Z 379.95,A -85,B 0,C 180,E1 -17187.865,E2 -17187.865} C_VEL
LIN {X 0,Y 282.511,Z 382.974,A -85,B 0,C 180,E1 -17190,E2 -17190} C_VEL
LIN {X 0,Y 282.383,Z 385.8,A -85,B 0,C 180,E1 -17192.853,E2 -17192.853} C_VEL
LIN {X 0,Y 282.335,Z 387.282,A -85,B 0,C 180,E1 -17195.715,E2 -17195.715} C_VEL
LIN {X 0,Y 282.258,Z 387.448,A -85,B 0,C 180,E1 -17198.592,E2 -17198.592} C_VEL
LIN {X 0,Y 282.494,Z 386.281,A -85,B 0,C 180,E1 -17201.48,E2 -17201.48} C_VEL
LIN {X 0,Y 283.169,Z 383.742,A -85,B 0,C 180,E1 -17204.371,E2 -17204.371} C_VEL
LIN {X 0,Y 284.119,Z 379.731,A -85,B 0,C 180,E1 -17207.268,E2 -17207.268} C_VEL
LIN {X 0,Y 285.635,Z 374.131,A -85,B 0,C 180,E1 -17210.149,E2 -17210.149} C_VEL
LIN {X 0,Y 287.408,Z 367.775,A -85,B 0,C 180,E1 -17212.652,E2 -17212.652} C_VEL
LIN {X 0,Y 289.645,Z 359.835,A -85,B 0,C 180,E1 -17215.127,E2 -17215.127} C_VEL
LIN {X 0,Y 291.891,Z 351.499,A -85,B 0,C 180,E1 -17217.224,E2 -17217.224} C_VEL
LIN {X 0,Y 294.428,Z 341.418,A -85,B 0,C 180,E1 -17219.297,E2 -17219.297} C_VEL
LIN {X 0,Y 296.901,Z 331.252,A -85,B 0,C 180,E1 -17220.988,E2 -17220.988} C_VEL
LIN {X 0,Y 299.29,Z 320.456,A -85,B 0,C 180,E1 -17222.456,E2 -17222.456} C_VEL
LIN {X 0,Y 301.664,Z 308.264,A -85,B 0,C 180,E1 -17223.795,E2 -17223.795} C_VEL
LIN {X 0,Y 303.759,Z 295.088,A -85,B 0,C 180,E1 -17224.934,E2 -17224.934} C_VEL
LIN {X 0,Y 305.491,Z 280.576,A -85,B 0,C 180,E1 -17225.868,E2 -17225.868} C_VEL
LIN {X 0,Y 306.796,Z 265.999,A -85,B 0,C 180,E1 -17226.505,E2 -17226.505} C_VEL
LIN {X 0,Y 307.725,Z 246.022,A -85,B 0,C 180,E1 -17227.024,E2 -17227.024} C_VEL
LIN {X 0,Y 310.417,Z 175.293,A -85,B 0,C 180,E1 -17228.637,E2 -17228.637} C_VEL
LIN {X 0,Y 303.044,Z 158.871,A -85,B 0,C 180,E1 -17230.107,E2 -17230.107} C_VEL
LIN {X 0,Y 294.687,Z 143.001,A -85,B 0,C 180,E1 -17231.816,E2 -17231.816} C_VEL
LIN {X 0,Y 287.382,Z 130.588,A -85,B 0,C 180,E1 -17233.383,E2 -17233.383} C_VEL
LIN {X 0,Y 285.264,Z 126.683,A -85,B 0,C 180,E1 -17233.904,E2 -17233.904} C_VEL
LIN {X 0,Y 284.255,Z 123.187,A -85,B 0,C 180,E1 -17235.501,E2 -17235.501} C_VEL
LIN {X 0,Y 284.209,Z 123.196,A -85,B 0,C 180,E1 -17236.847,E2 -17236.847} C_VEL
LIN {X 0,Y 283.54,Z 123.293,A -85,B 0,C 180,E1 -17238.03,E2 -17238.03} C_VEL
LIN {X 0,Y 280.708,Z 123.648,A -85,B 0,C 180,E1 -17239.958,E2 -17239.958} C_VEL
LIN {X 0,Y 278.316,Z 123.944,A -85,B 0,C 180,E1 -17241.524,E2 -17241.524} C_VEL
LIN {X 0,Y 277.299,Z 124.07,A -85,B 0,C 180,E1 -17242.737,E2 -17242.737} C_VEL
LIN {X 0,Y 277.22,Z 124.073,A -85,B 0,C 180,E1 -17243.148,E2 -17243.148} C_VEL
LIN {X 0,Y 277.254,Z 124.068,A -85,B 0,C 180,E1 -17246.773,E2 -17246.773} C_VEL
LIN {X 0,Y 277.263,Z 124.067,A -85,B 0,C 180,E1 -17249.538,E2 -17249.538} C_VEL
LIN {X 0,Y 277.293,Z 124.064,A -85,B 0,C 180,E1 -17252.857,E2 -17252.857} C_VEL
LIN {X 0,Y 277.284,Z 124.071,A -85,B 0,C 180,E1 -17256.075,E2 -17256.075} C_VEL
LIN {X 0,Y 277.33,Z 124.058,A -85,B 0,C 180,E1 -17260.765,E2 -17260.765} C_VEL
LIN {X 0,Y 277.411,Z 124.049,A -85,B 0,C 180,E1 -17265.324,E2 -17265.324} C_VEL
LIN {X 0,Y 277.461,Z 124.044,A -85,B 0,C 180,E1 -17269.787,E2 -17269.787} C_VEL
LIN {X 0,Y 277.606,Z 124.027,A -85,B 0,C 180,E1 -17272.728,E2 -17272.728} C_VEL
LIN {X 0,Y 277.82,Z 124.004,A -85,B 0,C 180,E1 -17278.55,E2 -17278.55} C_VEL
LIN {X 0,Y 277.819,Z 123.989,A -85,B 0,C 180,E1 -17281.449,E2 -17281.449} C_VEL
LIN {X 0,Y 277.602,Z 124.02,A -85,B 0,C 180,E1 -17287.272,E2 -17287.272} C_VEL
LIN {X 0,Y 277.458,Z 124.042,A -85,B 0,C 180,E1 -17290.213,E2 -17290.213} C_VEL
LIN {X 0,Y 277.436,Z 124.049,A -85,B 0,C 180,E1 -17294.674,E2 -17294.674} C_VEL
LIN {X 0,Y 277.346,Z 124.058,A -85,B 0,C 180,E1 -17299.234,E2 -17299.234} C_VEL
LIN {X 0,Y 277.32,Z 124.057,A -85,B 0,C 180,E1 -17304.17,E2 -17304.17} C_VEL
LIN {X 0,Y 277.327,Z 124.061,A -85,B 0,C 180,E1 -17307.505,E2 -17307.505} C_VEL
LIN {X 0,Y 277.273,Z 124.071,A -85,B 0,C 180,E1 -17310.481,E2 -17310.481} C_VEL
LIN {X 0,Y 277.248,Z 124.075,A -85,B 0,C 180,E1 -17313.895,E2 -17313.895} C_VEL
LIN {X 0,Y 277.266,Z 124.073,A -85,B 0,C 180,E1 -17317.469,E2 -17317.469} C_VEL
LIN {X 0,Y 277.21,Z 124.065,A -85,B 0,C 180,E1 -17321.236,E2 -17321.236} C_VEL
LIN {X 0,Y 277.201,Z 124.064,A -85,B 0,C 180,E1 -17325.226,E2 -17325.226} C_VEL
LIN {X 0,Y 277.246,Z 124.279,A -85,B 0,C 180,E1 -17326.373,E2 -17326.373} C_VEL
LIN {X 0,Y 279.515,Z 131.64,A -85,B 0,C 180,E1 -17329.515,E2 -17329.515} C_VEL
LIN {X 0,Y 280.92,Z 136.613,A -85,B 0,C 180,E1 -17331.425,E2 -17331.425} C_VEL
LIN {X 0,Y 283.264,Z 140.826,A -85,B 0,C 180,E1 -17331.974,E2 -17331.974} C_VEL
LIN {X 0,Y 289.066,Z 151.33,A -85,B 0,C 180,E1 -17333.281,E2 -17333.281} C_VEL
LIN {X 0,Y 296.878,Z 167.099,A -85,B 0,C 180,E1 -17334.972,E2 -17334.972} C_VEL
LIN {X 0,Y 302.168,Z 179.115,A -85,B 0,C 180,E1 -17336.085,E2 -17336.085} C_VEL
LIN {X 0,Y 304.044,Z 190.848,A -85,B 0,C 180,E1 -17336.68,E2 -17336.68} C_VEL
LIN {X 0,Y 300.735,Z 274.858,A -85,B 0,C 180,E1 -17338.67,E2 -17338.67} C_VEL
LIN {X 0,Y 299.37,Z 289.396,A -85,B 0,C 180,E1 -17339.247,E2 -17339.247} C_VEL
LIN {X 0,Y 297.538,Z 303.3,A -85,B 0,C 180,E1 -17340.067,E2 -17340.067} C_VEL
LIN {X 0,Y 295.209,Z 317.116,A -85,B 0,C 180,E1 -17341.178,E2 -17341.178} C_VEL
LIN {X 0,Y 292.794,Z 329.5,A -85,B 0,C 180,E1 -17342.48,E2 -17342.48} C_VEL
LIN {X 0,Y 290.036,Z 342.004,A -85,B 0,C 180,E1 -17344.14,E2 -17344.14} C_VEL
LIN {X 0,Y 287.409,Z 352.246,A -85,B 0,C 180,E1 -17345.821,E2 -17345.821} C_VEL
LIN {X 0,Y 284.627,Z 362.455,A -85,B 0,C 180,E1 -17347.88,E2 -17347.88} C_VEL
LIN {X 0,Y 282.215,Z 370.92,A -85,B 0,C 180,E1 -17349.976,E2 -17349.976} C_VEL
LIN {X 0,Y 279.871,Z 379.022,A -85,B 0,C 180,E1 -17352.462,E2 -17352.462} C_VEL
LIN {X 0,Y 278.434,Z 384.741,A -85,B 0,C 180,E1 -17354.631,E2 -17354.631} C_VEL
LIN {X 0,Y 277.161,Z 389.408,A -85,B 0,C 180,E1 -17356.808,E2 -17356.808} C_VEL
LIN {X 0,Y 276.048,Z 394.266,A -85,B 0,C 180,E1 -17359.734,E2 -17359.734} C_VEL
LIN {X 0,Y 275.447,Z 397.653,A -85,B 0,C 180,E1 -17362.67,E2 -17362.67} C_VEL
LIN {X 0,Y 275.207,Z 399.662,A -85,B 0,C 180,E1 -17365.606,E2 -17365.606} C_VEL
LIN {X 0,Y 275.237,Z 400.332,A -85,B 0,C 180,E1 -17368.537,E2 -17368.537} C_VEL
LIN {X 0,Y 275.246,Z 399.661,A -85,B 0,C 180,E1 -17371.463,E2 -17371.463} C_VEL
LIN {X 0,Y 275.205,Z 397.63,A -85,B 0,C 180,E1 -17374.394,E2 -17374.394} C_VEL
LIN {X 0,Y 275.388,Z 394.186,A -85,B 0,C 180,E1 -17377.331,E2 -17377.331} C_VEL
LIN {X 0,Y 275.876,Z 389.222,A -85,B 0,C 180,E1 -17380.272,E2 -17380.272} C_VEL
LIN {X 0,Y 276.555,Z 384.424,A -85,B 0,C 180,E1 -17382.474,E2 -17382.474} C_VEL
LIN {X 0,Y 277.757,Z 377.469,A -85,B 0,C 180,E1 -17385.031,E2 -17385.031} C_VEL
LIN {X 0,Y 279.202,Z 368.819,A -85,B 0,C 180,E1 -17387.581,E2 -17387.581} C_VEL
LIN {X 0,Y 280.977,Z 359.785,A -85,B 0,C 180,E1 -17389.735,E2 -17389.735} C_VEL
LIN {X 0,Y 282.683,Z 350.801,A -85,B 0,C 180,E1 -17391.513,E2 -17391.513} C_VEL
LIN {X 0,Y 284.759,Z 340.085,A -85,B 0,C 180,E1 -17393.259,E2 -17393.259} C_VEL
LIN {X 0,Y 286.761,Z 328.115,A -85,B 0,C 180,E1 -17394.85,E2 -17394.85} C_VEL
LIN {X 0,Y 288.729,Z 315.482,A -85,B 0,C 180,E1 -17396.179,E2 -17396.179} C_VEL
LIN {X 0,Y 290.437,Z 302.071,A -85,B 0,C 180,E1 -17397.274,E2 -17397.274} C_VEL
LIN {X 0,Y 291.853,Z 288.229,A -85,B 0,C 180,E1 -17398.104,E2 -17398.104} C_VEL
LIN {X 0,Y 292.902,Z 273.76,A -85,B 0,C 180,E1 -17398.678,E2 -17398.678} C_VEL
LIN {X 0,Y 295.635,Z 186.129,A -85,B 0,C 180,E1 -17400.79,E2 -17400.79} C_VEL
LIN {X 0,Y 292.254,Z 164.84,A -85,B 0,C 180,E1 -17401.729,E2 -17401.729} C_VEL
LIN {X 0,Y 284.904,Z 147.03,A -85,B 0,C 180,E1 -17403.06,E2 -17403.06} C_VEL
LIN {X 0,Y 280.423,Z 136.756,A -85,B 0,C 180,E1 -17403.937,E2 -17403.937} C_VEL
LIN {X 0,Y 277.741,Z 125.819,A -85,B 0,C 180,E1 -17407.697,E2 -17407.697} C_VEL
LIN {X 0,Y 277.273,Z 124.076,A -85,B 0,C 180,E1 -17408.397,E2 -17408.397} C_VEL
LIN {X 0,Y 277.232,Z 124.076,A -85,B 0,C 180,E1 -17412.679,E2 -17412.679} C_VEL
LIN {X 0,Y 277.262,Z 124.07,A -85,B 0,C 180,E1 -17416.812,E2 -17416.812} C_VEL
LIN {X 0,Y 277.265,Z 124.058,A -85,B 0,C 180,E1 -17420.677,E2 -17420.677} C_VEL
LIN {X 0,Y 277.303,Z 124.066,A -85,B 0,C 180,E1 -17424.344,E2 -17424.344} C_VEL
LIN {X 0,Y 277.243,Z 124.075,A -85,B 0,C 180,E1 -17427.836,E2 -17427.836} C_VEL
LIN {X 0,Y 277.29,Z 124.066,A -85,B 0,C 180,E1 -17431.213,E2 -17431.213} C_VEL
LIN {X 0,Y 277.314,Z 124.065,A -85,B 0,C 180,E1 -17434.48,E2 -17434.48} C_VEL
LIN {X 0,Y 277.284,Z 124.069,A -85,B 0,C 180,E1 -17437.655,E2 -17437.655} C_VEL
LIN {X 0,Y 277.344,Z 124.057,A -85,B 0,C 180,E1 -17440.766,E2 -17440.766} C_VEL
LIN {X 0,Y 277.434,Z 124.049,A -85,B 0,C 180,E1 -17445.326,E2 -17445.326} C_VEL
LIN {X 0,Y 277.505,Z 124.04,A -85,B 0,C 180,E1 -17449.789,E2 -17449.789} C_VEL
LIN {X 0,Y 277.643,Z 124.021,A -85,B 0,C 180,E1 -17452.729,E2 -17452.729} C_VEL
LIN {X 0,Y 277.819,Z 124.003,A -85,B 0,C 180,E1 -17458.551,E2 -17458.551} C_VEL
LIN {X 0,Y 277.819,Z 123.992,A -85,B 0,C 180,E1 -17461.45,E2 -17461.45} C_VEL
LIN {X 0,Y 277.611,Z 124.027,A -85,B 0,C 180,E1 -17467.272,E2 -17467.272} C_VEL
LIN {X 0,Y 277.459,Z 124.037,A -85,B 0,C 180,E1 -17470.213,E2 -17470.213} C_VEL
LIN {X 0,Y 277.434,Z 124.049,A -85,B 0,C 180,E1 -17474.674,E2 -17474.674} C_VEL
LIN {X 0,Y 277.345,Z 124.055,A -85,B 0,C 180,E1 -17479.234,E2 -17479.234} C_VEL
LIN {X 0,Y 277.329,Z 124.056,A -85,B 0,C 180,E1 -17483.921,E2 -17483.921} C_VEL
LIN {X 0,Y 277.323,Z 124.066,A -85,B 0,C 180,E1 -17487.505,E2 -17487.505} C_VEL
LIN {X 0,Y 277.272,Z 124.067,A -85,B 0,C 180,E1 -17490.482,E2 -17490.482} C_VEL
LIN {X 0,Y 277.247,Z 124.074,A -85,B 0,C 180,E1 -17493.896,E2 -17493.896} C_VEL
LIN {X 0,Y 277.265,Z 124.068,A -85,B 0,C 180,E1 -17497.47,E2 -17497.47} C_VEL
LIN {X 0,Y 277.21,Z 124.074,A -85,B 0,C 180,E1 -17501.237,E2 -17501.237} C_VEL
LIN {X 0,Y 277.217,Z 124.074,A -85,B 0,C 180,E1 -17505.224,E2 -17505.224} C_VEL
LIN {X 0,Y 277.223,Z 124.071,A -85,B 0,C 180,E1 -17509.513,E2 -17509.513} C_VEL
LIN {X 0,Y 277.265,Z 124.064,A -85,B 0,C 180,E1 -17512.531,E2 -17512.531} C_VEL
LIN {X 0,Y 277.248,Z 124.076,A -85,B 0,C 180,E1 -17516.105,E2 -17516.105} C_VEL
LIN {X 0,Y 277.275,Z 124.071,A -85,B 0,C 180,E1 -17520.796,E2 -17520.796} C_VEL
LIN {X 0,Y 277.283,Z 124.193,A -85,B 0,C 180,E1 -17521.005,E2 -17521.005} C_VEL
LIN {X 0,Y 277.854,Z 126.396,A -85,B 0,C 180,E1 -17521.831,E2 -17521.831} C_VEL
LIN {X 0,Y 287.275,Z 146.211,A -85,B 0,C 180,E1 -17523.568,E2 -17523.568} C_VEL
LIN {X 0,Y 294.544,Z 164.032,A -85,B 0,C 180,E1 -17524.871,E2 -17524.871} C_VEL
LIN {X 0,Y 296.202,Z 168.945,A -85,B 0,C 180,E1 -17525.18,E2 -17525.18} C_VEL
LIN {X 0,Y 293.154,Z 263.014,A -85,B 0,C 180,E1 -17527.445,E2 -17527.445} C_VEL
LIN {X 0,Y 292.321,Z 276.755,A -85,B 0,C 180,E1 -17528.028,E2 -17528.028} C_VEL
LIN {X 0,Y 291.091,Z 290.266,A -85,B 0,C 180,E1 -17528.86,E2 -17528.86} C_VEL
LIN {X 0,Y 289.44,Z 303.443,A -85,B 0,C 180,E1 -17529.942,E2 -17529.942} C_VEL
LIN {X 0,Y 287.558,Z 316.14,A -85,B 0,C 180,E1 -17531.29,E2 -17531.29} C_VEL
LIN {X 0,Y 285.621,Z 327.685,A -85,B 0,C 180,E1 -17532.826,E2 -17532.826} C_VEL
LIN {X 0,Y 283.674,Z 338.27,A -85,B 0,C 180,E1 -17534.554,E2 -17534.554} C_VEL
LIN {X 0,Y 281.619,Z 348.928,A -85,B 0,C 180,E1 -17536.691,E2 -17536.691} C_VEL
LIN {X 0,Y 279.992,Z 357.428,A -85,B 0,C 180,E1 -17538.783,E2 -17538.783} C_VEL
LIN {X 0,Y 278.522,Z 364.646,A -85,B 0,C 180,E1 -17540.926,E2 -17540.926} C_VEL
LIN {X 0,Y 277.189,Z 371.559,A -85,B 0,C 180,E1 -17543.449,E2 -17543.449} C_VEL
LIN {X 0,Y 276.306,Z 376.359,A -85,B 0,C 180,E1 -17545.624,E2 -17545.624} C_VEL
LIN {X 0,Y 275.831,Z 380.259,A -85,B 0,C 180,E1 -17547.81,E2 -17547.81} C_VEL
LIN {X 0,Y 275.425,Z 383.247,A -85,B 0,C 180,E1 -17550,E2 -17550} C_VEL
LIN {X 0,Y 275.288,Z 386.033,A -85,B 0,C 180,E1 -17552.927,E2 -17552.927} C_VEL
LIN {X 0,Y 275.227,Z 387.476,A -85,B 0,C 180,E1 -17555.863,E2 -17555.863} C_VEL
LIN {X 0,Y 275.164,Z 387.602,A -85,B 0,C 180,E1 -17558.815,E2 -17558.815} C_VEL
LIN {X 0,Y 275.47,Z 386.392,A -85,B 0,C 180,E1 -17561.777,E2 -17561.777} C_VEL
LIN {X 0,Y 276.204,Z 383.753,A -85,B 0,C 180,E1 -17564.779,E2 -17564.779} C_VEL
LIN {X 0,Y 277.216,Z 379.74,A -85,B 0,C 180,E1 -17567.712,E2 -17567.712} C_VEL
LIN {X 0,Y 278.834,Z 374.093,A -85,B 0,C 180,E1 -17570.663,E2 -17570.663} C_VEL
LIN {X 0,Y 280.718,Z 367.686,A -85,B 0,C 180,E1 -17573.223,E2 -17573.223} C_VEL
LIN {X 0,Y 283.12,Z 359.69,A -85,B 0,C 180,E1 -17575.748,E2 -17575.748} C_VEL
LIN {X 0,Y 285.449,Z 351.288,A -85,B 0,C 180,E1 -17577.891,E2 -17577.891} C_VEL
LIN {X 0,Y 288.142,Z 341.134,A -85,B 0,C 180,E1 -17580.001,E2 -17580.001} C_VEL
LIN {X 0,Y 290.757,Z 330.879,A -85,B 0,C 180,E1 -17581.717,E2 -17581.717} C_VEL
LIN {X 0,Y 293.243,Z 319.737,A -85,B 0,C 180,E1 -17583.246,E2 -17583.246} C_VEL
LIN {X 0,Y 295.738,Z 307.62,A -85,B 0,C 180,E1 -17584.567,E2 -17584.567} C_VEL
LIN {X 0,Y 297.881,Z 294.13,A -85,B 0,C 180,E1 -17585.728,E2 -17585.728} C_VEL
LIN {X 0,Y 299.629,Z 279.998,A -85,B 0,C 180,E1 -17586.631,E2 -17586.631} C_VEL
LIN {X 0,Y 300.943,Z 265.474,A -85,B 0,C 180,E1 -17587.262,E2 -17587.262} C_VEL
LIN {X 0,Y 301.917,Z 243.827,A -85,B 0,C 180,E1 -17587.825,E2 -17587.825} C_VEL
LIN {X 0,Y 304.539,Z 177.367,A -85,B 0,C 180,E1 -17589.366,E2 -17589.366} C_VEL
LIN {X 0,Y 298.001,Z 162.687,A -85,B 0,C 180,E1 -17590.722,E2 -17590.722} C_VEL
LIN {X 0,Y 289.989,Z 147.314,A -85,B 0,C 180,E1 -17592.424,E2 -17592.424} C_VEL
LIN {X 0,Y 282.835,Z 135.104,A -85,B 0,C 180,E1 -17594.016,E2 -17594.016} C_VEL
LIN {X 0,Y 279.646,Z 129.885,A -85,B 0,C 180,E1 -17594.757,E2 -17594.757} C_VEL
LIN {X 0,Y 277.996,Z 126.848,A -85,B 0,C 180,E1 -17595.216,E2 -17595.216} C_VEL
LIN {X 0,Y 277.174,Z 124.071,A -85,B 0,C 180,E1 -17596.522,E2 -17596.522} C_VEL
LIN {X 0,Y 277.191,Z 124.06,A -85,B 0,C 180,E1 -17600.664,E2 -17600.664} C_VEL
LIN {X 0,Y 277.22,Z 124.073,A -85,B 0,C 180,E1 -17603.148,E2 -17603.148} C_VEL
LIN {X 0,Y 276.566,Z 124.155,A -85,B 0,C 180,E1 -17604.36,E2 -17604.36} C_VEL
LIN {X 0,Y 273.722,Z 124.51,A -85,B 0,C 180,E1 -17606.335,E2 -17606.335} C_VEL
LIN {X 0,Y 271.3,Z 124.814,A -85,B 0,C 180,E1 -17607.94,E2 -17607.94} C_VEL
LIN {X 0,Y 270.257,Z 124.943,A -85,B 0,C 180,E1 -17609.184,E2 -17609.184} C_VEL
LIN {X 0,Y 270.17,Z 124.95,A -85,B 0,C 180,E1 -17609.606,E2 -17609.606} C_VEL
LIN {X 0,Y 270.224,Z 124.95,A -85,B 0,C 180,E1 -17612.163,E2 -17612.163} C_VEL
LIN {X 0,Y 270.229,Z 124.95,A -85,B 0,C 180,E1 -17615.542,E2 -17615.542} C_VEL
LIN {X 0,Y 270.28,Z 124.942,A -85,B 0,C 180,E1 -17620.243,E2 -17620.243} C_VEL
LIN {X 0,Y 270.379,Z 124.927,A -85,B 0,C 180,E1 -17624.934,E2 -17624.934} C_VEL
LIN {X 0,Y 270.413,Z 124.925,A -85,B 0,C 180,E1 -17629.518,E2 -17629.518} C_VEL
LIN {X 0,Y 270.567,Z 124.901,A -85,B 0,C 180,E1 -17632.537,E2 -17632.537} C_VEL
LIN {X 0,Y 270.785,Z 124.881,A -85,B 0,C 180,E1 -17638.513,E2 -17638.513} C_VEL
LIN {X 0,Y 270.785,Z 124.865,A -85,B 0,C 180,E1 -17641.487,E2 -17641.487} C_VEL
LIN {X 0,Y 270.564,Z 124.898,A -85,B 0,C 180,E1 -17647.462,E2 -17647.462} C_VEL
LIN {X 0,Y 270.411,Z 124.917,A -85,B 0,C 180,E1 -17650.482,E2 -17650.482} C_VEL
LIN {X 0,Y 270.404,Z 124.919,A -85,B 0,C 180,E1 -17655.064,E2 -17655.064} C_VEL
LIN {X 0,Y 270.303,Z 124.931,A -85,B 0,C 180,E1 -17659.755,E2 -17659.755} C_VEL
LIN {X 0,Y 270.275,Z 124.932,A -85,B 0,C 180,E1 -17664.585,E2 -17664.585} C_VEL
LIN {X 0,Y 270.271,Z 124.938,A -85,B 0,C 180,E1 -17667.908,E2 -17667.908} C_VEL
LIN {X 0,Y 270.185,Z 124.951,A -85,B 0,C 180,E1 -17671.348,E2 -17671.348} C_VEL
LIN {X 0,Y 270.202,Z 124.948,A -85,B 0,C 180,E1 -17674.905,E2 -17674.905} C_VEL
LIN {X 0,Y 270.198,Z 124.934,A -85,B 0,C 180,E1 -17678.71,E2 -17678.71} C_VEL
LIN {X 0,Y 270.172,Z 124.956,A -85,B 0,C 180,E1 -17682.558,E2 -17682.558} C_VEL
LIN {X 0,Y 270.167,Z 124.964,A -85,B 0,C 180,E1 -17685.139,E2 -17685.139} C_VEL
LIN {X 0,Y 272.821,Z 133.663,A -85,B 0,C 180,E1 -17689.01,E2 -17689.01} C_VEL
LIN {X 0,Y 273.576,Z 136.386,A -85,B 0,C 180,E1 -17690.062,E2 -17690.062} C_VEL
LIN {X 0,Y 276.155,Z 140.734,A -85,B 0,C 180,E1 -17690.698,E2 -17690.698} C_VEL
LIN {X 0,Y 284.028,Z 154.885,A -85,B 0,C 180,E1 -17692.562,E2 -17692.562} C_VEL
LIN {X 0,Y 291.932,Z 171.059,A -85,B 0,C 180,E1 -17694.346,E2 -17694.346} C_VEL
LIN {X 0,Y 296.729,Z 182.063,A -85,B 0,C 180,E1 -17695.396,E2 -17695.396} C_VEL
LIN {X 0,Y 298.275,Z 191.251,A -85,B 0,C 180,E1 -17695.891,E2 -17695.891} C_VEL
LIN {X 0,Y 294.823,Z 275.218,A -85,B 0,C 180,E1 -17697.917,E2 -17697.917} C_VEL
LIN {X 0,Y 293.434,Z 289.579,A -85,B 0,C 180,E1 -17698.505,E2 -17698.505} C_VEL
LIN {X 0,Y 291.439,Z 303.957,A -85,B 0,C 180,E1 -17699.374,E2 -17699.374} C_VEL
LIN {X 0,Y 289.047,Z 317.594,A -85,B 0,C 180,E1 -17700.504,E2 -17700.504} C_VEL
LIN {X 0,Y 286.532,Z 329.854,A -85,B 0,C 180,E1 -17701.825,E2 -17701.825} C_VEL
LIN {X 0,Y 283.664,Z 342.251,A -85,B 0,C 180,E1 -17703.515,E2 -17703.515} C_VEL
LIN {X 0,Y 280.932,Z 352.428,A -85,B 0,C 180,E1 -17705.226,E2 -17705.226} C_VEL
LIN {X 0,Y 278.066,Z 362.558,A -85,B 0,C 180,E1 -17707.329,E2 -17707.329} C_VEL
LIN {X 0,Y 275.548,Z 370.98,A -85,B 0,C 180,E1 -17709.47,E2 -17709.47} C_VEL
LIN {X 0,Y 273.068,Z 379.039,A -85,B 0,C 180,E1 -17712.01,E2 -17712.01} C_VEL
LIN {X 0,Y 271.538,Z 384.735,A -85,B 0,C 180,E1 -17714.231,E2 -17714.231} C_VEL
LIN {X 0,Y 269.852,Z 390.73,A -85,B 0,C 180,E1 -17717.21,E2 -17717.21} C_VEL
LIN {X 0,Y 269.011,Z 394.197,A -85,B 0,C 180,E1 -17719.462,E2 -17719.462} C_VEL
LIN {X 0,Y 268.368,Z 397.554,A -85,B 0,C 180,E1 -17722.476,E2 -17722.476} C_VEL
LIN {X 0,Y 268.109,Z 399.528,A -85,B 0,C 180,E1 -17725.489,E2 -17725.489} C_VEL
LIN {X 0,Y 268.164,Z 400.166,A -85,B 0,C 180,E1 -17728.498,E2 -17728.498} C_VEL
LIN {X 0,Y 268.172,Z 399.463,A -85,B 0,C 180,E1 -17731.501,E2 -17731.501} C_VEL
LIN {X 0,Y 268.108,Z 397.401,A -85,B 0,C 180,E1 -17734.51,E2 -17734.51} C_VEL
LIN {X 0,Y 268.315,Z 393.927,A -85,B 0,C 180,E1 -17737.525,E2 -17737.525} C_VEL
LIN {X 0,Y 268.849,Z 388.931,A -85,B 0,C 180,E1 -17740.544,E2 -17740.544} C_VEL
LIN {X 0,Y 269.581,Z 384.098,A -85,B 0,C 180,E1 -17742.802,E2 -17742.802} C_VEL
LIN {X 0,Y 270.867,Z 377.106,A -85,B 0,C 180,E1 -17745.423,E2 -17745.423} C_VEL
LIN {X 0,Y 272.115,Z 369.781,A -85,B 0,C 180,E1 -17747.665,E2 -17747.665} C_VEL
LIN {X 0,Y 273.902,Z 360.971,A -85,B 0,C 180,E1 -17749.875,E2 -17749.875} C_VEL
LIN {X 0,Y 276.028,Z 350.285,A -85,B 0,C 180,E1 -17752.058,E2 -17752.058} C_VEL
LIN {X 0,Y 278.215,Z 339.501,A -85,B 0,C 180,E1 -17753.839,E2 -17753.839} C_VEL
LIN {X 0,Y 280.225,Z 327.84,A -85,B 0,C 180,E1 -17755.415,E2 -17755.415} C_VEL
LIN {X 0,Y 282.313,Z 314.681,A -85,B 0,C 180,E1 -17756.821,E2 -17756.821} C_VEL
LIN {X 0,Y 284.143,Z 301.099,A -85,B 0,C 180,E1 -17757.93,E2 -17757.93} C_VEL
LIN {X 0,Y 285.598,Z 286.822,A -85,B 0,C 180,E1 -17758.776,E2 -17758.776} C_VEL
LIN {X 0,Y 286.581,Z 272.946,A -85,B 0,C 180,E1 -17759.321,E2 -17759.321} C_VEL
LIN {X 0,Y 289.332,Z 186.807,A -85,B 0,C 180,E1 -17761.439,E2 -17761.439} C_VEL
LIN {X 0,Y 286.276,Z 167.307,A -85,B 0,C 180,E1 -17762.324,E2 -17762.324} C_VEL
LIN {X 0,Y 278.2,Z 147.721,A -85,B 0,C 180,E1 -17763.85,E2 -17763.85} C_VEL
LIN {X 0,Y 273.14,Z 136.602,A -85,B 0,C 180,E1 -17764.86,E2 -17764.86} C_VEL
LIN {X 0,Y 270.767,Z 127.062,A -85,B 0,C 180,E1 -17768.265,E2 -17768.265} C_VEL
LIN {X 0,Y 270.211,Z 124.953,A -85,B 0,C 180,E1 -17769.102,E2 -17769.102} C_VEL
LIN {X 0,Y 270.188,Z 124.955,A -85,B 0,C 180,E1 -17773.254,E2 -17773.254} C_VEL
LIN {X 0,Y 270.247,Z 124.945,A -85,B 0,C 180,E1 -17777.457,E2 -17777.457} C_VEL
LIN {X 0,Y 270.244,Z 124.929,A -85,B 0,C 180,E1 -17781.381,E2 -17781.381} C_VEL
LIN {X 0,Y 270.214,Z 124.951,A -85,B 0,C 180,E1 -17785.097,E2 -17785.097} C_VEL
LIN {X 0,Y 270.199,Z 124.954,A -85,B 0,C 180,E1 -17789.131,E2 -17789.131} C_VEL
LIN {X 0,Y 270.264,Z 124.942,A -85,B 0,C 180,E1 -17792.145,E2 -17792.145} C_VEL
LIN {X 0,Y 270.276,Z 124.936,A -85,B 0,C 180,E1 -17795.519,E2 -17795.519} C_VEL
LIN {X 0,Y 270.301,Z 124.936,A -85,B 0,C 180,E1 -17800.245,E2 -17800.245} C_VEL
LIN {X 0,Y 270.402,Z 124.927,A -85,B 0,C 180,E1 -17804.936,E2 -17804.936} C_VEL
LIN {X 0,Y 270.441,Z 124.92,A -85,B 0,C 180,E1 -17809.519,E2 -17809.519} C_VEL
LIN {X 0,Y 270.602,Z 124.899,A -85,B 0,C 180,E1 -17812.539,E2 -17812.539} C_VEL
LIN {X 0,Y 270.785,Z 124.88,A -85,B 0,C 180,E1 -17818.513,E2 -17818.513} C_VEL
LIN {X 0,Y 270.785,Z 124.868,A -85,B 0,C 180,E1 -17821.487,E2 -17821.487} C_VEL
LIN {X 0,Y 270.571,Z 124.904,A -85,B 0,C 180,E1 -17827.463,E2 -17827.463} C_VEL
LIN {X 0,Y 270.412,Z 124.915,A -85,B 0,C 180,E1 -17830.483,E2 -17830.483} C_VEL
LIN {X 0,Y 270.403,Z 124.925,A -85,B 0,C 180,E1 -17835.065,E2 -17835.065} C_VEL
LIN {X 0,Y 270.302,Z 124.936,A -85,B 0,C 180,E1 -17839.756,E2 -17839.756} C_VEL
LIN {X 0,Y 270.274,Z 124.933,A -85,B 0,C 180,E1 -17844.586,E2 -17844.586} C_VEL
LIN {X 0,Y 270.271,Z 124.943,A -85,B 0,C 180,E1 -17847.909,E2 -17847.909} C_VEL
LIN {X 0,Y 270.184,Z 124.947,A -85,B 0,C 180,E1 -17851.349,E2 -17851.349} C_VEL
LIN {X 0,Y 270.201,Z 124.954,A -85,B 0,C 180,E1 -17854.906,E2 -17854.906} C_VEL
LIN {X 0,Y 270.198,Z 124.951,A -85,B 0,C 180,E1 -17858.711,E2 -17858.711} C_VEL
LIN {X 0,Y 270.172,Z 124.957,A -85,B 0,C 180,E1 -17863.251,E2 -17863.251} C_VEL
LIN {X 0,Y 270.175,Z 124.955,A -85,B 0,C 180,E1 -17867.443,E2 -17867.443} C_VEL
LIN {X 0,Y 270.208,Z 124.934,A -85,B 0,C 180,E1 -17871.375,E2 -17871.375} C_VEL
LIN {X 0,Y 270.202,Z 124.951,A -85,B 0,C 180,E1 -17875.095,E2 -17875.095} C_VEL
LIN {X 0,Y 270.219,Z 124.952,A -85,B 0,C 180,E1 -17879.591,E2 -17879.591} C_VEL
LIN {X 0,Y 270.261,Z 125.043,A -85,B 0,C 180,E1 -17880.292,E2 -17880.292} C_VEL
LIN {X 0,Y 270.63,Z 126.607,A -85,B 0,C 180,E1 -17880.896,E2 -17880.896} C_VEL
LIN {X 0,Y 280.13,Z 146.133,A -85,B 0,C 180,E1 -17882.716,E2 -17882.716} C_VEL
LIN {X 0,Y 287.367,Z 163.374,A -85,B 0,C 180,E1 -17884.063,E2 -17884.063} C_VEL
LIN {X 0,Y 289.896,Z 170.021,A -85,B 0,C 180,E1 -17884.531,E2 -17884.531} C_VEL
LIN {X 0,Y 286.797,Z 263.225,A -85,B 0,C 180,E1 -17886.824,E2 -17886.824} C_VEL
LIN {X 0,Y 285.94,Z 276.898,A -85,B 0,C 180,E1 -17887.416,E2 -17887.416} C_VEL
LIN {X 0,Y 284.662,Z 290.417,A -85,B 0,C 180,E1 -17888.264,E2 -17888.264} C_VEL
LIN {X 0,Y 283.061,Z 302.723,A -85,B 0,C 180,E1 -17889.28,E2 -17889.28} C_VEL
LIN {X 0,Y 281.108,Z 315.59,A -85,B 0,C 180,E1 -17890.655,E2 -17890.655} C_VEL
LIN {X 0,Y 278.887,Z 328.424,A -85,B 0,C 180,E1 -17892.398,E2 -17892.398} C_VEL
LIN {X 0,Y 276.875,Z 338.912,A -85,B 0,C 180,E1 -17894.165,E2 -17894.165} C_VEL
LIN {X 0,Y 274.776,Z 349.328,A -85,B 0,C 180,E1 -17896.315,E2 -17896.315} C_VEL
LIN {X 0,Y 273.067,Z 357.923,A -85,B 0,C 180,E1 -17898.495,E2 -17898.495} C_VEL
LIN {X 0,Y 271.294,Z 366.19,A -85,B 0,C 180,E1 -17901.058,E2 -17901.058} C_VEL
LIN {X 0,Y 270.152,Z 371.944,A -85,B 0,C 180,E1 -17903.277,E2 -17903.277} C_VEL
LIN {X 0,Y 269.243,Z 376.697,A -85,B 0,C 180,E1 -17905.509,E2 -17905.509} C_VEL
LIN {X 0,Y 268.744,Z 380.558,A -85,B 0,C 180,E1 -17907.752,E2 -17907.752} C_VEL
LIN {X 0,Y 268.341,Z 383.519,A -85,B 0,C 180,E1 -17910,E2 -17910} C_VEL
LIN {X 0,Y 268.195,Z 386.265,A -85,B 0,C 180,E1 -17913.004,E2 -17913.004} C_VEL
LIN {X 0,Y 268.134,Z 387.669,A -85,B 0,C 180,E1 -17916.018,E2 -17916.018} C_VEL
LIN {X 0,Y 268.086,Z 387.756,A -85,B 0,C 180,E1 -17919.05,E2 -17919.05} C_VEL
LIN {X 0,Y 268.425,Z 386.496,A -85,B 0,C 180,E1 -17922.091,E2 -17922.091} C_VEL
LIN {X 0,Y 269.211,Z 383.851,A -85,B 0,C 180,E1 -17925.133,E2 -17925.133} C_VEL
LIN {X 0,Y 270.33,Z 379.75,A -85,B 0,C 180,E1 -17928.178,E2 -17928.178} C_VEL
LIN {X 0,Y 272.073,Z 374.056,A -85,B 0,C 180,E1 -17931.201,E2 -17931.201} C_VEL
LIN {X 0,Y 274.069,Z 367.598,A -85,B 0,C 180,E1 -17933.821,E2 -17933.821} C_VEL
LIN {X 0,Y 276.616,Z 359.546,A -85,B 0,C 180,E1 -17936.399,E2 -17936.399} C_VEL
LIN {X 0,Y 279.067,Z 351.081,A -85,B 0,C 180,E1 -17938.587,E2 -17938.587} C_VEL
LIN {X 0,Y 281.907,Z 340.84,A -85,B 0,C 180,E1 -17940.735,E2 -17940.735} C_VEL
LIN {X 0,Y 284.644,Z 330.494,A -85,B 0,C 180,E1 -17942.481,E2 -17942.481} C_VEL
LIN {X 0,Y 287.511,Z 317.782,A -85,B 0,C 180,E1 -17944.209,E2 -17944.209} C_VEL
LIN {X 0,Y 290.169,Z 305.134,A -85,B 0,C 180,E1 -17945.541,E2 -17945.541} C_VEL
LIN {X 0,Y 292.253,Z 292.037,A -85,B 0,C 180,E1 -17946.633,E2 -17946.633} C_VEL
LIN {X 0,Y 293.904,Z 278.745,A -85,B 0,C 180,E1 -17947.459,E2 -17947.459} C_VEL
LIN {X 0,Y 295.151,Z 264.871,A -85,B 0,C 180,E1 -17948.053,E2 -17948.053} C_VEL
LIN {X 0,Y 296.382,Z 237.124,A -85,B 0,C 180,E1 -17948.759,E2 -17948.759} C_VEL
LIN {X 0,Y 298.715,Z 179.312,A -85,B 0,C 180,E1 -17950.126,E2 -17950.126} C_VEL
LIN {X 0,Y 291.326,Z 163.028,A -85,B 0,C 180,E1 -17951.724,E2 -17951.724} C_VEL
LIN {X 0,Y 283.079,Z 147.699,A -85,B 0,C 180,E1 -17953.561,E2 -17953.561} C_VEL
LIN {X 0,Y 275.601,Z 135.037,A -85,B 0,C 180,E1 -17955.329,E2 -17955.329} C_VEL
LIN {X 0,Y 272.897,Z 130.837,A -85,B 0,C 180,E1 -17955.992,E2 -17955.992} C_VEL
LIN {X 0,Y 270.807,Z 127.162,A -85,B 0,C 180,E1 -17956.551,E2 -17956.551} C_VEL
LIN {X 0,Y 270.157,Z 124.959,A -85,B 0,C 180,E1 -17957.65,E2 -17957.65} C_VEL
LIN {X 0,Y 270.153,Z 124.943,A -85,B 0,C 180,E1 -17961.364,E2 -17961.364} C_VEL
LIN {X 0,Y 270.199,Z 124.952,A -85,B 0,C 180,E1 -17965.094,E2 -17965.094} C_VEL
LIN {X 0,Y 270.186,Z 124.952,A -85,B 0,C 180,E1 -17969.136,E2 -17969.136} C_VEL
LIN {X 0,Y 270.17,Z 124.95,A -85,B 0,C 180,E1 -17969.606,E2 -17969.606} C_VEL
LIN {X 0,Y 269.501,Z 125.036,A -85,B 0,C 180,E1 -17970.85,E2 -17970.85} C_VEL
LIN {X 0,Y 266.661,Z 125.388,A -85,B 0,C 180,E1 -17972.876,E2 -17972.876} C_VEL
LIN {X 0,Y 264.256,Z 125.688,A -85,B 0,C 180,E1 -17974.524,E2 -17974.524} C_VEL
LIN {X 0,Y 263.228,Z 125.822,A -85,B 0,C 180,E1 -17975.801,E2 -17975.801} C_VEL
LIN {X 0,Y 263.146,Z 125.828,A -85,B 0,C 180,E1 -17976.233,E2 -17976.233} C_VEL
LIN {X 0,Y 263.245,Z 125.819,A -85,B 0,C 180,E1 -17979.692,E2 -17979.692} C_VEL
LIN {X 0,Y 263.325,Z 125.808,A -85,B 0,C 180,E1 -17984.52,E2 -17984.52} C_VEL
LIN {X 0,Y 263.356,Z 125.805,A -85,B 0,C 180,E1 -17989.233,E2 -17989.233} C_VEL
LIN {X 0,Y 263.53,Z 125.774,A -85,B 0,C 180,E1 -17992.337,E2 -17992.337} C_VEL
LIN {X 0,Y 263.75,Z 125.757,A -85,B 0,C 180,E1 -17998.473,E2 -17998.473} C_VEL
LIN {X 0,Y 263.75,Z 125.741,A -85,B 0,C 180,E1 -18001.527,E2 -18001.527} C_VEL
LIN {X 0,Y 263.528,Z 125.776,A -85,B 0,C 180,E1 -18007.663,E2 -18007.663} C_VEL
LIN {X 0,Y 263.354,Z 125.794,A -85,B 0,C 180,E1 -18010.766,E2 -18010.766} C_VEL
LIN {X 0,Y 263.352,Z 125.793,A -85,B 0,C 180,E1 -18015.478,E2 -18015.478} C_VEL
LIN {X 0,Y 263.265,Z 125.803,A -85,B 0,C 180,E1 -18020.306,E2 -18020.306} C_VEL
LIN {X 0,Y 263.21,Z 125.811,A -85,B 0,C 180,E1 -18025.291,E2 -18025.291} C_VEL
LIN {X 0,Y 263.167,Z 125.818,A -85,B 0,C 180,E1 -18028.731,E2 -18028.731} C_VEL
LIN {X 0,Y 263.134,Z 125.825,A -85,B 0,C 180,E1 -18032.288,E2 -18032.288} C_VEL
LIN {X 0,Y 263.163,Z 125.823,A -85,B 0,C 180,E1 -18035.982,E2 -18035.982} C_VEL
LIN {X 0,Y 263.105,Z 125.81,A -85,B 0,C 180,E1 -18039.872,E2 -18039.872} C_VEL
LIN {X 0,Y 263.104,Z 125.896,A -85,B 0,C 180,E1 -18043.916,E2 -18043.916} C_VEL
LIN {X 0,Y 266.181,Z 135.829,A -85,B 0,C 180,E1 -18048.537,E2 -18048.537} C_VEL
LIN {X 0,Y 268.879,Z 140.54,A -85,B 0,C 180,E1 -18049.289,E2 -18049.289} C_VEL
LIN {X 0,Y 273.219,Z 148.127,A -85,B 0,C 180,E1 -18050.403,E2 -18050.403} C_VEL
LIN {X 0,Y 279.371,Z 159.119,A -85,B 0,C 180,E1 -18051.899,E2 -18051.899} C_VEL
LIN {X 0,Y 288.058,Z 177.183,A -85,B 0,C 180,E1 -18053.93,E2 -18053.93} C_VEL
LIN {X 0,Y 291.362,Z 185.182,A -85,B 0,C 180,E1 -18054.691,E2 -18054.691} C_VEL
LIN {X 0,Y 292.544,Z 193.562,A -85,B 0,C 180,E1 -18055.124,E2 -18055.124} C_VEL
LIN {X 0,Y 289.094,Z 274.432,A -85,B 0,C 180,E1 -18057.099,E2 -18057.099} C_VEL
LIN {X 0,Y 287.648,Z 289.004,A -85,B 0,C 180,E1 -18057.692,E2 -18057.692} C_VEL
LIN {X 0,Y 285.768,Z 302.365,A -85,B 0,C 180,E1 -18058.492,E2 -18058.492} C_VEL
LIN {X 0,Y 283.57,Z 314.561,A -85,B 0,C 180,E1 -18059.464,E2 -18059.464} C_VEL
LIN {X 0,Y 280.912,Z 327.373,A -85,B 0,C 180,E1 -18060.8,E2 -18060.8} C_VEL
LIN {X 0,Y 277.988,Z 339.982,A -85,B 0,C 180,E1 -18062.486,E2 -18062.486} C_VEL
LIN {X 0,Y 275.057,Z 350.681,A -85,B 0,C 180,E1 -18064.255,E2 -18064.255} C_VEL
LIN {X 0,Y 271.99,Z 361.117,A -85,B 0,C 180,E1 -18066.39,E2 -18066.39} C_VEL
LIN {X 0,Y 269.302,Z 369.744,A -85,B 0,C 180,E1 -18068.57,E2 -18068.57} C_VEL
LIN {X 0,Y 266.631,Z 378.04,A -85,B 0,C 180,E1 -18071.162,E2 -18071.162} C_VEL
LIN {X 0,Y 264.668,Z 384.725,A -85,B 0,C 180,E1 -18073.81,E2 -18073.81} C_VEL
LIN {X 0,Y 262.887,Z 390.677,A -85,B 0,C 180,E1 -18076.865,E2 -18076.865} C_VEL
LIN {X 0,Y 261.993,Z 394.128,A -85,B 0,C 180,E1 -18079.177,E2 -18079.177} C_VEL
LIN {X 0,Y 261.309,Z 397.451,A -85,B 0,C 180,E1 -18082.271,E2 -18082.271} C_VEL
LIN {X 0,Y 261.017,Z 399.39,A -85,B 0,C 180,E1 -18085.367,E2 -18085.367} C_VEL
LIN {X 0,Y 261.07,Z 399.996,A -85,B 0,C 180,E1 -18088.457,E2 -18088.457} C_VEL
LIN {X 0,Y 261.095,Z 399.798,A -85,B 0,C 180,E1 -18090,E2 -18090} C_VEL
LIN {X 0,Y 261.041,Z 398.392,A -85,B 0,C 180,E1 -18093.086,E2 -18093.086} C_VEL
LIN {X 0,Y 261.133,Z 395.604,A -85,B 0,C 180,E1 -18096.18,E2 -18096.18} C_VEL
LIN {X 0,Y 261.483,Z 391.352,A -85,B 0,C 180,E1 -18099.28,E2 -18099.28} C_VEL
LIN {X 0,Y 262.264,Z 385.509,A -85,B 0,C 180,E1 -18102.379,E2 -18102.379} C_VEL
LIN {X 0,Y 263.487,Z 378.921,A -85,B 0,C 180,E1 -18105.073,E2 -18105.073} C_VEL
LIN {X 0,Y 265.045,Z 370.728,A -85,B 0,C 180,E1 -18107.754,E2 -18107.754} C_VEL
LIN {X 0,Y 266.849,Z 362.145,A -85,B 0,C 180,E1 -18110.022,E2 -18110.022} C_VEL
LIN {X 0,Y 269.005,Z 351.738,A -85,B 0,C 180,E1 -18112.261,E2 -18112.261} C_VEL
LIN {X 0,Y 271.463,Z 340.095,A -85,B 0,C 180,E1 -18114.267,E2 -18114.267} C_VEL
LIN {X 0,Y 273.539,Z 328.448,A -85,B 0,C 180,E1 -18115.898,E2 -18115.898} C_VEL
LIN {X 0,Y 275.683,Z 315.653,A -85,B 0,C 180,E1 -18117.314,E2 -18117.314} C_VEL
LIN {X 0,Y 277.542,Z 302.384,A -85,B 0,C 180,E1 -18118.449,E2 -18118.449} C_VEL
LIN {X 0,Y 279.125,Z 287.996,A -85,B 0,C 180,E1 -18119.353,E2 -18119.353} C_VEL
LIN {X 0,Y 280.221,Z 273.599,A -85,B 0,C 180,E1 -18119.95,E2 -18119.95} C_VEL
LIN {X 0,Y 283.112,Z 187.843,A -85,B 0,C 180,E1 -18122.101,E2 -18122.101} C_VEL
LIN {X 0,Y 280.366,Z 169.847,A -85,B 0,C 180,E1 -18122.938,E2 -18122.938} C_VEL
LIN {X 0,Y 272.357,Z 150.43,A -85,B 0,C 180,E1 -18124.511,E2 -18124.511} C_VEL
LIN {X 0,Y 265.877,Z 136.396,A -85,B 0,C 180,E1 -18125.857,E2 -18125.857} C_VEL
LIN {X 0,Y 263.464,Z 127.128,A -85,B 0,C 180,E1 -18129.323,E2 -18129.323} C_VEL
LIN {X 0,Y 263.13,Z 125.836,A -85,B 0,C 180,E1 -18129.868,E2 -18129.868} C_VEL
LIN {X 0,Y 263.137,Z 125.832,A -85,B 0,C 180,E1 -18133.981,E2 -18133.981} C_VEL
LIN {X 0,Y 263.209,Z 125.823,A -85,B 0,C 180,E1 -18138.385,E2 -18138.385} C_VEL
LIN {X 0,Y 263.203,Z 125.817,A -85,B 0,C 180,E1 -18143.23,E2 -18143.23} C_VEL
LIN {X 0,Y 263.183,Z 125.822,A -85,B 0,C 180,E1 -18145.89,E2 -18145.89} C_VEL
LIN {X 0,Y 263.15,Z 125.829,A -85,B 0,C 180,E1 -18149.507,E2 -18149.507} C_VEL
LIN {X 0,Y 263.193,Z 125.826,A -85,B 0,C 180,E1 -18153.003,E2 -18153.003} C_VEL
LIN {X 0,Y 263.183,Z 125.819,A -85,B 0,C 180,E1 -18156.387,E2 -18156.387} C_VEL
LIN {X 0,Y 263.263,Z 125.813,A -85,B 0,C 180,E1 -18159.694,E2 -18159.694} C_VEL
LIN {X 0,Y 263.35,Z 125.807,A -85,B 0,C 180,E1 -18164.522,E2 -18164.522} C_VEL
LIN {X 0,Y 263.373,Z 125.801,A -85,B 0,C 180,E1 -18169.235,E2 -18169.235} C_VEL
LIN {X 0,Y 263.564,Z 125.778,A -85,B 0,C 180,E1 -18172.338,E2 -18172.338} C_VEL
LIN {X 0,Y 263.75,Z 125.756,A -85,B 0,C 180,E1 -18178.473,E2 -18178.473} C_VEL
LIN {X 0,Y 263.75,Z 125.743,A -85,B 0,C 180,E1 -18181.527,E2 -18181.527} C_VEL
LIN {X 0,Y 263.533,Z 125.782,A -85,B 0,C 180,E1 -18187.663,E2 -18187.663} C_VEL
LIN {X 0,Y 263.354,Z 125.794,A -85,B 0,C 180,E1 -18190.767,E2 -18190.767} C_VEL
LIN {X 0,Y 263.35,Z 125.804,A -85,B 0,C 180,E1 -18195.478,E2 -18195.478} C_VEL
LIN {X 0,Y 263.268,Z 125.814,A -85,B 0,C 180,E1 -18200.307,E2 -18200.307} C_VEL
LIN {X 0,Y 263.208,Z 125.812,A -85,B 0,C 180,E1 -18205.292,E2 -18205.292} C_VEL
LIN {X 0,Y 263.179,Z 125.827,A -85,B 0,C 180,E1 -18208.73,E2 -18208.73} C_VEL
LIN {X 0,Y 263.133,Z 125.826,A -85,B 0,C 180,E1 -18212.289,E2 -18212.289} C_VEL
LIN {X 0,Y 263.181,Z 125.821,A -85,B 0,C 180,E1 -18216.763,E2 -18216.763} C_VEL
LIN {X 0,Y 263.125,Z 125.826,A -85,B 0,C 180,E1 -18221.594,E2 -18221.594} C_VEL
LIN {X 0,Y 263.129,Z 125.827,A -85,B 0,C 180,E1 -18226.018,E2 -18226.018} C_VEL
LIN {X 0,Y 263.106,Z 125.822,A -85,B 0,C 180,E1 -18230.128,E2 -18230.128} C_VEL
LIN {X 0,Y 263.164,Z 125.831,A -85,B 0,C 180,E1 -18234.019,E2 -18234.019} C_VEL
LIN {X 0,Y 263.129,Z 125.833,A -85,B 0,C 180,E1 -18237.712,E2 -18237.712} C_VEL
LIN {X 0,Y 263.169,Z 125.858,A -85,B 0,C 180,E1 -18239.51,E2 -18239.51} C_VEL
LIN {X 0,Y 263.463,Z 127.1,A -85,B 0,C 180,E1 -18239.915,E2 -18239.915} C_VEL
LIN {X 0,Y 271.394,Z 142.774,A -85,B 0,C 180,E1 -18241.504,E2 -18241.504} C_VEL
LIN {X 0,Y 277.862,Z 157.12,A -85,B 0,C 180,E1 -18242.761,E2 -18242.761} C_VEL
LIN {X 0,Y 283.599,Z 171.621,A -85,B 0,C 180,E1 -18243.867,E2 -18243.867} C_VEL
LIN {X 0,Y 280.552,Z 261.885,A -85,B 0,C 180,E1 -18246.127,E2 -18246.127} C_VEL
LIN {X 0,Y 279.721,Z 275.368,A -85,B 0,C 180,E1 -18246.69,E2 -18246.69} C_VEL
LIN {X 0,Y 278.387,Z 289.426,A -85,B 0,C 180,E1 -18247.553,E2 -18247.553} C_VEL
LIN {X 0,Y 276.767,Z 301.977,A -85,B 0,C 180,E1 -18248.591,E2 -18248.591} C_VEL
LIN {X 0,Y 274.678,Z 315.032,A -85,B 0,C 180,E1 -18249.988,E2 -18249.988} C_VEL
LIN {X 0,Y 272.663,Z 326.822,A -85,B 0,C 180,E1 -18251.594,E2 -18251.594} C_VEL
LIN {X 0,Y 270.519,Z 337.611,A -85,B 0,C 180,E1 -18253.395,E2 -18253.395} C_VEL
LIN {X 0,Y 268.225,Z 348.277,A -85,B 0,C 180,E1 -18255.587,E2 -18255.587} C_VEL
LIN {X 0,Y 266.399,Z 357.077,A -85,B 0,C 180,E1 -18257.816,E2 -18257.816} C_VEL
LIN {X 0,Y 264.573,Z 365.52,A -85,B 0,C 180,E1 -18260.444,E2 -18260.444} C_VEL
LIN {X 0,Y 263.12,Z 372.33,A -85,B 0,C 180,E1 -18263.097,E2 -18263.097} C_VEL
LIN {X 0,Y 262.183,Z 377.035,A -85,B 0,C 180,E1 -18265.388,E2 -18265.388} C_VEL
LIN {X 0,Y 261.66,Z 380.852,A -85,B 0,C 180,E1 -18267.691,E2 -18267.691} C_VEL
LIN {X 0,Y 261.259,Z 383.792,A -85,B 0,C 180,E1 -18270,E2 -18270} C_VEL
LIN {X 0,Y 261.106,Z 386.497,A -85,B 0,C 180,E1 -18273.086,E2 -18273.086} C_VEL
LIN {X 0,Y 261.026,Z 387.863,A -85,B 0,C 180,E1 -18276.183,E2 -18276.183} C_VEL
LIN {X 0,Y 261.006,Z 387.902,A -85,B 0,C 180,E1 -18279.298,E2 -18279.298} C_VEL
LIN {X 0,Y 261.397,Z 386.592,A -85,B 0,C 180,E1 -18282.421,E2 -18282.421} C_VEL
LIN {X 0,Y 262.249,Z 383.904,A -85,B 0,C 180,E1 -18285.545,E2 -18285.545} C_VEL
LIN {X 0,Y 263.454,Z 379.76,A -85,B 0,C 180,E1 -18288.67,E2 -18288.67} C_VEL
LIN {X 0,Y 265.345,Z 374.02,A -85,B 0,C 180,E1 -18291.766,E2 -18291.766} C_VEL
LIN {X 0,Y 267.458,Z 367.513,A -85,B 0,C 180,E1 -18294.448,E2 -18294.448} C_VEL
LIN {X 0,Y 270.157,Z 359.406,A -85,B 0,C 180,E1 -18297.081,E2 -18297.081} C_VEL
LIN {X 0,Y 272.738,Z 350.878,A -85,B 0,C 180,E1 -18299.314,E2 -18299.314} C_VEL
LIN {X 0,Y 275.71,Z 340.525,A -85,B 0,C 180,E1 -18301.504,E2 -18301.504} C_VEL
LIN {X 0,Y 278.624,Z 330.083,A -85,B 0,C 180,E1 -18303.273,E2 -18303.273} C_VEL
LIN {X 0,Y 281.277,Z 318.654,A -85,B 0,C 180,E1 -18304.864,E2 -18304.864} C_VEL
LIN {X 0,Y 284.011,Z 306.213,A -85,B 0,C 180,E1 -18306.214,E2 -18306.214} C_VEL
LIN {X 0,Y 286.157,Z 293.371,A -85,B 0,C 180,E1 -18307.324,E2 -18307.324} C_VEL
LIN {X 0,Y 287.956,Z 279.613,A -85,B 0,C 180,E1 -18308.212,E2 -18308.212} C_VEL
LIN {X 0,Y 289.268,Z 265.804,A -85,B 0,C 180,E1 -18308.824,E2 -18308.824} C_VEL
LIN {X 0,Y 290.388,Z 242.929,A -85,B 0,C 180,E1 -18309.432,E2 -18309.432} C_VEL
LIN {X 0,Y 292.99,Z 181.477,A -85,B 0,C 180,E1 -18310.904,E2 -18310.904} C_VEL
LIN {X 0,Y 286.078,Z 166.329,A -85,B 0,C 180,E1 -18312.459,E2 -18312.459} C_VEL
LIN {X 0,Y 278.565,Z 152.184,A -85,B 0,C 180,E1 -18314.203,E2 -18314.203} C_VEL
LIN {X 0,Y 271.647,Z 140.287,A -85,B 0,C 180,E1 -18315.902,E2 -18315.902} C_VEL
LIN {X 0,Y 265.798,Z 131.221,A -85,B 0,C 180,E1 -18317.411,E2 -18317.411} C_VEL
LIN {X 0,Y 263.45,Z 127.32,A -85,B 0,C 180,E1 -18318.106,E2 -18318.106} C_VEL
LIN {X 0,Y 263.115,Z 125.82,A -85,B 0,C 180,E1 -18318.894,E2 -18318.894} C_VEL
LIN {X 0,Y 263.152,Z 125.828,A -85,B 0,C 180,E1 -18323.246,E2 -18323.246} C_VEL
LIN {X 0,Y 263.153,Z 125.83,A -85,B 0,C 180,E1 -18325.885,E2 -18325.885} C_VEL
LIN {X 0,Y 263.122,Z 125.828,A -85,B 0,C 180,E1 -18329.587,E2 -18329.587} C_VEL
LIN {X 0,Y 263.142,Z 125.825,A -85,B 0,C 180,E1 -18332.997,E2 -18332.997} C_VEL
LIN {X 0,Y 263.146,Z 125.828,A -85,B 0,C 180,E1 -18336.233,E2 -18336.233} C_VEL
LIN {X 0,Y 262.482,Z 125.913,A -85,B 0,C 180,E1 -18337.512,E2 -18337.512} C_VEL
LIN {X 0,Y 259.639,Z 126.269,A -85,B 0,C 180,E1 -18339.596,E2 -18339.596} C_VEL
LIN {X 0,Y 257.248,Z 126.557,A -85,B 0,C 180,E1 -18341.291,E2 -18341.291} C_VEL
LIN {X 0,Y 256.258,Z 126.679,A -85,B 0,C 180,E1 -18342.605,E2 -18342.605} C_VEL
LIN {X 0,Y 256.195,Z 126.689,A -85,B 0,C 180,E1 -18343.05,E2 -18343.05} C_VEL
LIN {X 0,Y 256.29,Z 126.677,A -85,B 0,C 180,E1 -18347.327,E2 -18347.327} C_VEL
LIN {X 0,Y 256.436,Z 126.653,A -85,B 0,C 180,E1 -18350.622,E2 -18350.622} C_VEL
LIN {X 0,Y 256.462,Z 126.665,A -85,B 0,C 180,E1 -18353.707,E2 -18353.707} C_VEL
LIN {X 0,Y 256.713,Z 126.634,A -85,B 0,C 180,E1 -18358.431,E2 -18358.431} C_VEL
LIN {X 0,Y 256.712,Z 126.617,A -85,B 0,C 180,E1 -18361.569,E2 -18361.569} C_VEL
LIN {X 0,Y 256.459,Z 126.649,A -85,B 0,C 180,E1 -18366.293,E2 -18366.293} C_VEL
LIN {X 0,Y 256.428,Z 126.667,A -85,B 0,C 180,E1 -18369.465,E2 -18369.465} C_VEL
LIN {X 0,Y 256.257,Z 126.688,A -85,B 0,C 180,E1 -18374.29,E2 -18374.29} C_VEL
LIN {X 0,Y 256.212,Z 126.686,A -85,B 0,C 180,E1 -18377.562,E2 -18377.562} C_VEL
LIN {X 0,Y 256.158,Z 126.687,A -85,B 0,C 180,E1 -18381.119,E2 -18381.119} C_VEL
LIN {X 0,Y 256.19,Z 126.685,A -85,B 0,C 180,E1 -18385.138,E2 -18385.138} C_VEL
LIN {X 0,Y 256.105,Z 126.701,A -85,B 0,C 180,E1 -18389.601,E2 -18389.601} C_VEL
LIN {X 0,Y 256.077,Z 126.708,A -85,B 0,C 180,E1 -18393.291,E2 -18393.291} C_VEL
LIN {X 0,Y 256.115,Z 126.708,A -85,B 0,C 180,E1 -18397.27,E2 -18397.27} C_VEL
LIN {X 0,Y 256.054,Z 126.698,A -85,B 0,C 180,E1 -18401.203,E2 -18401.203} C_VEL
LIN {X 0,Y 256.068,Z 126.841,A -85,B 0,C 180,E1 -18402.605,E2 -18402.605} C_VEL
LIN {X 0,Y 258.286,Z 133.933,A -85,B 0,C 180,E1 -18406.143,E2 -18406.143} C_VEL
LIN {X 0,Y 258.882,Z 135.845,A -85,B 0,C 180,E1 -18406.987,E2 -18406.987} C_VEL
LIN {X 0,Y 261.495,Z 140.2,A -85,B 0,C 180,E1 -18407.734,E2 -18407.734} C_VEL
LIN {X 0,Y 268.204,Z 151.39,A -85,B 0,C 180,E1 -18409.544,E2 -18409.544} C_VEL
LIN {X 0,Y 275.203,Z 164.295,A -85,B 0,C 180,E1 -18411.327,E2 -18411.327} C_VEL
LIN {X 0,Y 283.388,Z 181.609,A -85,B 0,C 180,E1 -18413.316,E2 -18413.316} C_VEL
LIN {X 0,Y 285.98,Z 187.957,A -85,B 0,C 180,E1 -18413.938,E2 -18413.938} C_VEL
LIN {X 0,Y 286.906,Z 194.109,A -85,B 0,C 180,E1 -18414.277,E2 -18414.277} C_VEL
LIN {X 0,Y 283.286,Z 274.799,A -85,B 0,C 180,E1 -18416.282,E2 -18416.282} C_VEL
LIN {X 0,Y 281.806,Z 289.19,A -85,B 0,C 180,E1 -18416.885,E2 -18416.885} C_VEL
LIN {X 0,Y 279.78,Z 303.021,A -85,B 0,C 180,E1 -18417.738,E2 -18417.738} C_VEL
LIN {X 0,Y 277.193,Z 316.793,A -85,B 0,C 180,E1 -18418.896,E2 -18418.896} C_VEL
LIN {X 0,Y 274.423,Z 329.148,A -85,B 0,C 180,E1 -18420.251,E2 -18420.251} C_VEL
LIN {X 0,Y 271.588,Z 340.764,A -85,B 0,C 180,E1 -18421.874,E2 -18421.874} C_VEL
LIN {X 0,Y 268.686,Z 350.873,A -85,B 0,C 180,E1 -18423.598,E2 -18423.598} C_VEL
LIN {X 0,Y 265.464,Z 361.251,A -85,B 0,C 180,E1 -18425.773,E2 -18425.773} C_VEL
LIN {X 0,Y 262.686,Z 369.828,A -85,B 0,C 180,E1 -18428.003,E2 -18428.003} C_VEL
LIN {X 0,Y 259.883,Z 378.068,A -85,B 0,C 180,E1 -18430.654,E2 -18430.654} C_VEL
LIN {X 0,Y 257.817,Z 384.711,A -85,B 0,C 180,E1 -18433.368,E2 -18433.368} C_VEL
LIN {X 0,Y 255.939,Z 390.626,A -85,B 0,C 180,E1 -18436.502,E2 -18436.502} C_VEL
LIN {X 0,Y 254.992,Z 394.061,A -85,B 0,C 180,E1 -18438.876,E2 -18438.876} C_VEL
LIN {X 0,Y 254.246,Z 397.345,A -85,B 0,C 180,E1 -18442.055,E2 -18442.055} C_VEL
LIN {X 0,Y 253.925,Z 399.249,A -85,B 0,C 180,E1 -18445.237,E2 -18445.237} C_VEL
LIN {X 0,Y 253.978,Z 399.825,A -85,B 0,C 180,E1 -18448.414,E2 -18448.414} C_VEL
LIN {X 0,Y 254.024,Z 399.614,A -85,B 0,C 180,E1 -18450,E2 -18450} C_VEL
LIN {X 0,Y 253.939,Z 398.178,A -85,B 0,C 180,E1 -18453.173,E2 -18453.173} C_VEL
LIN {X 0,Y 254.043,Z 395.361,A -85,B 0,C 180,E1 -18456.353,E2 -18456.353} C_VEL
LIN {X 0,Y 254.45,Z 391.076,A -85,B 0,C 180,E1 -18459.539,E2 -18459.539} C_VEL
LIN {X 0,Y 255.292,Z 385.199,A -85,B 0,C 180,E1 -18462.723,E2 -18462.723} C_VEL
LIN {X 0,Y 256.599,Z 378.574,A -85,B 0,C 180,E1 -18465.488,E2 -18465.488} C_VEL
LIN {X 0,Y 258.2,Z 370.324,A -85,B 0,C 180,E1 -18468.241,E2 -18468.241} C_VEL
LIN {X 0,Y 260.128,Z 361.692,A -85,B 0,C 180,E1 -18470.562,E2 -18470.562} C_VEL
LIN {X 0,Y 262.387,Z 351.214,A -85,B 0,C 180,E1 -18472.853,E2 -18472.853} C_VEL
LIN {X 0,Y 264.723,Z 340.684,A -85,B 0,C 180,E1 -18474.717,E2 -18474.717} C_VEL
LIN {X 0,Y 266.796,Z 329.549,A -85,B 0,C 180,E1 -18476.341,E2 -18476.341} C_VEL
LIN {X 0,Y 269.062,Z 316.62,A -85,B 0,C 180,E1 -18477.833,E2 -18477.833} C_VEL
LIN {X 0,Y 270.98,Z 303.666,A -85,B 0,C 180,E1 -18478.99,E2 -18478.99} C_VEL
LIN {X 0,Y 272.593,Z 289.78,A -85,B 0,C 180,E1 -18479.915,E2 -18479.915} C_VEL
LIN {X 0,Y 273.796,Z 275.362,A -85,B 0,C 180,E1 -18480.568,E2 -18480.568} C_VEL
LIN {X 0,Y 275.319,Z 237.632,A -85,B 0,C 180,E1 -18481.552,E2 -18481.552} C_VEL
LIN {X 0,Y 276.928,Z 188.929,A -85,B 0,C 180,E1 -18482.791,E2 -18482.791} C_VEL
LIN {X 0,Y 274.515,Z 172.514,A -85,B 0,C 180,E1 -18483.571,E2 -18483.571} C_VEL
LIN {X 0,Y 267.238,Z 154.696,A -85,B 0,C 180,E1 -18485.059,E2 -18485.059} C_VEL
LIN {X 0,Y 259.92,Z 139.227,A -85,B 0,C 180,E1 -18486.586,E2 -18486.586} C_VEL
LIN {X 0,Y 258.649,Z 136.3,A -85,B 0,C 180,E1 -18486.881,E2 -18486.881} C_VEL
LIN {X 0,Y 256.071,Z 126.712,A -85,B 0,C 180,E1 -18490.717,E2 -18490.717} C_VEL
LIN {X 0,Y 256.071,Z 126.711,A -85,B 0,C 180,E1 -18494.473,E2 -18494.473} C_VEL
LIN {X 0,Y 256.13,Z 126.704,A -85,B 0,C 180,E1 -18498.812,E2 -18498.812} C_VEL
LIN {X 0,Y 256.153,Z 126.693,A -85,B 0,C 180,E1 -18502.871,E2 -18502.871} C_VEL
LIN {X 0,Y 256.084,Z 126.704,A -85,B 0,C 180,E1 -18506.71,E2 -18506.71} C_VEL
LIN {X 0,Y 256.138,Z 126.7,A -85,B 0,C 180,E1 -18511.405,E2 -18511.405} C_VEL
LIN {X 0,Y 256.166,Z 126.692,A -85,B 0,C 180,E1 -18515.699,E2 -18515.699} C_VEL
LIN {X 0,Y 256.166,Z 126.7,A -85,B 0,C 180,E1 -18519.105,E2 -18519.105} C_VEL
LIN {X 0,Y 256.299,Z 126.683,A -85,B 0,C 180,E1 -18524.085,E2 -18524.085} C_VEL
LIN {X 0,Y 256.309,Z 126.678,A -85,B 0,C 180,E1 -18528.934,E2 -18528.934} C_VEL
LIN {X 0,Y 256.527,Z 126.655,A -85,B 0,C 180,E1 -18532.127,E2 -18532.127} C_VEL
LIN {X 0,Y 256.713,Z 126.633,A -85,B 0,C 180,E1 -18538.431,E2 -18538.431} C_VEL
LIN {X 0,Y 256.712,Z 126.618,A -85,B 0,C 180,E1 -18541.569,E2 -18541.569} C_VEL
LIN {X 0,Y 256.455,Z 126.662,A -85,B 0,C 180,E1 -18546.585,E2 -18546.585} C_VEL
LIN {X 0,Y 256.426,Z 126.655,A -85,B 0,C 180,E1 -18549.465,E2 -18549.465} C_VEL
LIN {X 0,Y 256.255,Z 126.689,A -85,B 0,C 180,E1 -18554.29,E2 -18554.29} C_VEL
LIN {X 0,Y 256.211,Z 126.682,A -85,B 0,C 180,E1 -18557.562,E2 -18557.562} C_VEL
LIN {X 0,Y 256.185,Z 126.698,A -85,B 0,C 180,E1 -18561.136,E2 -18561.136} C_VEL
LIN {X 0,Y 256.188,Z 126.685,A -85,B 0,C 180,E1 -18565.139,E2 -18565.139} C_VEL
LIN {X 0,Y 256.113,Z 126.704,A -85,B 0,C 180,E1 -18569.6,E2 -18569.6} C_VEL
LIN {X 0,Y 256.068,Z 126.711,A -85,B 0,C 180,E1 -18573.293,E2 -18573.293} C_VEL
LIN {X 0,Y 256.114,Z 126.7,A -85,B 0,C 180,E1 -18577.271,E2 -18577.271} C_VEL
LIN {X 0,Y 256.055,Z 126.708,A -85,B 0,C 180,E1 -18581.204,E2 -18581.204} C_VEL
LIN {X 0,Y 256.063,Z 126.707,A -85,B 0,C 180,E1 -18585.53,E2 -18585.53} C_VEL
LIN {X 0,Y 256.056,Z 126.711,A -85,B 0,C 180,E1 -18588.797,E2 -18588.797} C_VEL
LIN {X 0,Y 256.131,Z 126.698,A -85,B 0,C 180,E1 -18592.868,E2 -18592.868} C_VEL
LIN {X 0,Y 256.067,Z 126.716,A -85,B 0,C 180,E1 -18596.708,E2 -18596.708} C_VEL
LIN {X 0,Y 256.117,Z 126.913,A -85,B 0,C 180,E1 -18598.776,E2 -18598.776} C_VEL
LIN {X 0,Y 257.416,Z 130.026,A -85,B 0,C 180,E1 -18599.111,E2 -18599.111} C_VEL
LIN {X 0,Y 258.661,Z 131.859,A -85,B 0,C 180,E1 -18599.36,E2 -18599.36} C_VEL
LIN {X 0,Y 265.816,Z 145.975,A -85,B 0,C 180,E1 -18600.848,E2 -18600.848} C_VEL
LIN {X 0,Y 272.385,Z 160.619,A -85,B 0,C 180,E1 -18602.177,E2 -18602.177} C_VEL
LIN {X 0,Y 277.395,Z 173.435,A -85,B 0,C 180,E1 -18603.185,E2 -18603.185} C_VEL
LIN {X 0,Y 274.226,Z 263.341,A -85,B 0,C 180,E1 -18605.49,E2 -18605.49} C_VEL
LIN {X 0,Y 273.282,Z 277.144,A -85,B 0,C 180,E1 -18606.106,E2 -18606.106} C_VEL
LIN {X 0,Y 271.893,Z 290.685,A -85,B 0,C 180,E1 -18606.986,E2 -18606.986} C_VEL
LIN {X 0,Y 270.221,Z 302.997,A -85,B 0,C 180,E1 -18608.046,E2 -18608.046} C_VEL
LIN {X 0,Y 268.07,Z 315.883,A -85,B 0,C 180,E1 -18609.473,E2 -18609.473} C_VEL
LIN {X 0,Y 265.97,Z 327.553,A -85,B 0,C 180,E1 -18611.114,E2 -18611.114} C_VEL
LIN {X 0,Y 263.764,Z 338.245,A -85,B 0,C 180,E1 -18612.957,E2 -18612.957} C_VEL
LIN {X 0,Y 261.401,Z 348.832,A -85,B 0,C 180,E1 -18615.202,E2 -18615.202} C_VEL
LIN {X 0,Y 259.496,Z 357.567,A -85,B 0,C 180,E1 -18617.487,E2 -18617.487} C_VEL
LIN {X 0,Y 257.608,Z 365.952,A -85,B 0,C 180,E1 -18620.183,E2 -18620.183} C_VEL
LIN {X 0,Y 256.094,Z 372.712,A -85,B 0,C 180,E1 -18622.907,E2 -18622.907} C_VEL
LIN {X 0,Y 255.127,Z 377.371,A -85,B 0,C 180,E1 -18625.26,E2 -18625.26} C_VEL
LIN {X 0,Y 254.391,Z 382.206,A -85,B 0,C 180,E1 -18628.417,E2 -18628.417} C_VEL
LIN {X 0,Y 254.092,Z 385.566,A -85,B 0,C 180,E1 -18631.585,E2 -18631.585} C_VEL
LIN {X 0,Y 253.975,Z 387.555,A -85,B 0,C 180,E1 -18634.762,E2 -18634.762} C_VEL
LIN {X 0,Y 253.911,Z 388.213,A -85,B 0,C 180,E1 -18637.955,E2 -18637.955} C_VEL
LIN {X 0,Y 254.062,Z 387.534,A -85,B 0,C 180,E1 -18641.165,E2 -18641.165} C_VEL
LIN {X 0,Y 254.797,Z 385.499,A -85,B 0,C 180,E1 -18644.374,E2 -18644.374} C_VEL
LIN {X 0,Y 255.859,Z 382.055,A -85,B 0,C 180,E1 -18647.587,E2 -18647.587} C_VEL
LIN {X 0,Y 257.547,Z 377.089,A -85,B 0,C 180,E1 -18650.778,E2 -18650.778} C_VEL
LIN {X 0,Y 259.221,Z 372.259,A -85,B 0,C 180,E1 -18653.148,E2 -18653.148} C_VEL
LIN {X 0,Y 261.607,Z 365.25,A -85,B 0,C 180,E1 -18655.884,E2 -18655.884} C_VEL
LIN {X 0,Y 264.573,Z 356.534,A -85,B 0,C 180,E1 -18658.564,E2 -18658.564} C_VEL
LIN {X 0,Y 267.429,Z 347.382,A -85,B 0,C 180,E1 -18660.828,E2 -18660.828} C_VEL
LIN {X 0,Y 270.142,Z 338.236,A -85,B 0,C 180,E1 -18662.672,E2 -18662.672} C_VEL
LIN {X 0,Y 273.24,Z 327.294,A -85,B 0,C 180,E1 -18664.462,E2 -18664.462} C_VEL
LIN {X 0,Y 276.059,Z 315.259,A -85,B 0,C 180,E1 -18666.067,E2 -18666.067} C_VEL
LIN {X 0,Y 278.926,Z 301.898,A -85,B 0,C 180,E1 -18667.436,E2 -18667.436} C_VEL
LIN {X 0,Y 280.999,Z 288.896,A -85,B 0,C 180,E1 -18668.473,E2 -18668.473} C_VEL
LIN {X 0,Y 282.678,Z 275.155,A -85,B 0,C 180,E1 -18669.273,E2 -18669.273} C_VEL
LIN {X 0,Y 283.887,Z 260.666,A -85,B 0,C 180,E1 -18669.824,E2 -18669.824} C_VEL
LIN {X 0,Y 287.335,Z 183.68,A -85,B 0,C 180,E1 -18671.709,E2 -18671.709} C_VEL
LIN {X 0,Y 280.321,Z 168.372,A -85,B 0,C 180,E1 -18673.358,E2 -18673.358} C_VEL
LIN {X 0,Y 272.07,Z 152.981,A -85,B 0,C 180,E1 -18675.375,E2 -18675.375} C_VEL
LIN {X 0,Y 264.912,Z 141,A -85,B 0,C 180,E1 -18677.235,E2 -18677.235} C_VEL
LIN {X 0,Y 258.907,Z 131.819,A -85,B 0,C 180,E1 -18678.892,E2 -18678.892} C_VEL
LIN {X 0,Y 256.614,Z 128.743,A -85,B 0,C 180,E1 -18679.541,E2 -18679.541} C_VEL
LIN {X 0,Y 256.217,Z 127.608,A -85,B 0,C 180,E1 -18679.712,E2 -18679.712} C_VEL
LIN {X 0,Y 256.029,Z 126.694,A -85,B 0,C 180,E1 -18680.229,E2 -18680.229} C_VEL
LIN {X 0,Y 256.1,Z 126.71,A -85,B 0,C 180,E1 -18682.862,E2 -18682.862} C_VEL
LIN {X 0,Y 256.068,Z 126.707,A -85,B 0,C 180,E1 -18686.707,E2 -18686.707} C_VEL
LIN {X 0,Y 256.056,Z 126.706,A -85,B 0,C 180,E1 -18690.393,E2 -18690.393} C_VEL
LIN {X 0,Y 256.134,Z 126.701,A -85,B 0,C 180,E1 -18694.888,E2 -18694.888} C_VEL
LIN {X 0,Y 256.149,Z 126.701,A -85,B 0,C 180,E1 -18699.103,E2 -18699.103} C_VEL
LIN {X 0,Y 256.195,Z 126.689,A -85,B 0,C 180,E1 -18703.05,E2 -18703.05} C_VEL
LIN {X 0,Y 255.567,Z 126.776,A -85,B 0,C 180,E1 -18704.363,E2 -18704.363} C_VEL
LIN {X 0,Y 252.712,Z 127.132,A -85,B 0,C 180,E1 -18706.502,E2 -18706.502} C_VEL
LIN {X 0,Y 250.314,Z 127.428,A -85,B 0,C 180,E1 -18708.243,E2 -18708.243} C_VEL
LIN {X 0,Y 249.358,Z 127.545,A -85,B 0,C 180,E1 -18709.595,E2 -18709.595} C_VEL
LIN {X 0,Y 249.32,Z 127.542,A -85,B 0,C 180,E1 -18710.052,E2 -18710.052} C_VEL
LIN {X 0,Y 249.432,Z 127.54,A -85,B 0,C 180,E1 -18713.528,E2 -18713.528} C_VEL
LIN {X 0,Y 249.674,Z 127.511,A -85,B 0,C 180,E1 -18718.387,E2 -18718.387} C_VEL
LIN {X 0,Y 249.674,Z 127.494,A -85,B 0,C 180,E1 -18721.613,E2 -18721.613} C_VEL
LIN {X 0,Y 249.432,Z 127.524,A -85,B 0,C 180,E1 -18726.471,E2 -18726.471} C_VEL
LIN {X 0,Y 249.344,Z 127.547,A -85,B 0,C 180,E1 -18729.736,E2 -18729.736} C_VEL
LIN {X 0,Y 249.207,Z 127.563,A -85,B 0,C 180,E1 -18734.703,E2 -18734.703} C_VEL
LIN {X 0,Y 249.141,Z 127.574,A -85,B 0,C 180,E1 -18738.077,E2 -18738.077} C_VEL
LIN {X 0,Y 249.088,Z 127.57,A -85,B 0,C 180,E1 -18741.518,E2 -18741.518} C_VEL
LIN {X 0,Y 249.132,Z 127.565,A -85,B 0,C 180,E1 -18745.482,E2 -18745.482} C_VEL
LIN {X 0,Y 249.075,Z 127.573,A -85,B 0,C 180,E1 -18748.989,E2 -18748.989} C_VEL
LIN {X 0,Y 249.034,Z 127.581,A -85,B 0,C 180,E1 -18752.425,E2 -18752.425} C_VEL
LIN {X 0,Y 249.057,Z 127.582,A -85,B 0,C 180,E1 -18756.341,E2 -18756.341} C_VEL
LIN {X 0,Y 249.036,Z 127.689,A -85,B 0,C 180,E1 -18761.14,E2 -18761.14} C_VEL
LIN {X 0,Y 251.55,Z 135.646,A -85,B 0,C 180,E1 -18765.248,E2 -18765.248} C_VEL
LIN {X 0,Y 254.326,Z 140.161,A -85,B 0,C 180,E1 -18766.104,E2 -18766.104} C_VEL
LIN {X 0,Y 259.141,Z 147.916,A -85,B 0,C 180,E1 -18767.512,E2 -18767.512} C_VEL
LIN {X 0,Y 264.491,Z 157.217,A -85,B 0,C 180,E1 -18769.004,E2 -18769.004} C_VEL
LIN {X 0,Y 270.567,Z 168.44,A -85,B 0,C 180,E1 -18770.608,E2 -18770.608} C_VEL
LIN {X 0,Y 278.622,Z 185.791,A -85,B 0,C 180,E1 -18772.651,E2 -18772.651} C_VEL
LIN {X 0,Y 280.687,Z 190.942,A -85,B 0,C 180,E1 -18773.169,E2 -18773.169} C_VEL
LIN {X 0,Y 281.279,Z 196.03,A -85,B 0,C 180,E1 -18773.432,E2 -18773.432} C_VEL
LIN {X 0,Y 277.656,Z 274.053,A -85,B 0,C 180,E1 -18775.393,E2 -18775.393} C_VEL
LIN {X 0,Y 276.155,Z 288.636,A -85,B 0,C 180,E1 -18776.007,E2 -18776.007} C_VEL
LIN {X 0,Y 274.249,Z 301.444,A -85,B 0,C 180,E1 -18776.786,E2 -18776.786} C_VEL
LIN {X 0,Y 271.912,Z 313.768,A -85,B 0,C 180,E1 -18777.786,E2 -18777.786} C_VEL
LIN {X 0,Y 269,Z 326.671,A -85,B 0,C 180,E1 -18779.154,E2 -18779.154} C_VEL
LIN {X 0,Y 266.125,Z 338.015,A -85,B 0,C 180,E1 -18780.685,E2 -18780.685} C_VEL
LIN {X 0,Y 262.904,Z 349.124,A -85,B 0,C 180,E1 -18782.54,E2 -18782.54} C_VEL
LIN {X 0,Y 259.483,Z 359.762,A -85,B 0,C 180,E1 -18784.749,E2 -18784.749} C_VEL
LIN {X 0,Y 256.54,Z 368.56,A -85,B 0,C 180,E1 -18787.021,E2 -18787.021} C_VEL
LIN {X 0,Y 253.553,Z 377.011,A -85,B 0,C 180,E1 -18789.728,E2 -18789.728} C_VEL
LIN {X 0,Y 251.556,Z 382.93,A -85,B 0,C 180,E1 -18792.102,E2 -18792.102} C_VEL
LIN {X 0,Y 249.46,Z 389.267,A -85,B 0,C 180,E1 -18795.312,E2 -18795.312} C_VEL
LIN {X 0,Y 248.002,Z 393.991,A -85,B 0,C 180,E1 -18798.558,E2 -18798.558} C_VEL
LIN {X 0,Y 247.184,Z 397.235,A -85,B 0,C 180,E1 -18801.827,E2 -18801.827} C_VEL
LIN {X 0,Y 246.845,Z 399.139,A -85,B 0,C 180,E1 -18805.201,E2 -18805.201} C_VEL
LIN {X 0,Y 246.888,Z 399.655,A -85,B 0,C 180,E1 -18808.369,E2 -18808.369} C_VEL
LIN {X 0,Y 246.932,Z 399.43,A -85,B 0,C 180,E1 -18810,E2 -18810} C_VEL
LIN {X 0,Y 246.895,Z 398.867,A -85,B 0,C 180,E1 -18811.631,E2 -18811.631} C_VEL
LIN {X 0,Y 246.845,Z 396.716,A -85,B 0,C 180,E1 -18814.9,E2 -18814.9} C_VEL
LIN {X 0,Y 247.13,Z 393.147,A -85,B 0,C 180,E1 -18818.174,E2 -18818.174} C_VEL
LIN {X 0,Y 247.775,Z 388.05,A -85,B 0,C 180,E1 -18821.452,E2 -18821.452} C_VEL
LIN {X 0,Y 248.716,Z 383.113,A -85,B 0,C 180,E1 -18823.897,E2 -18823.897} C_VEL
LIN {X 0,Y 250.169,Z 375.948,A -85,B 0,C 180,E1 -18826.754,E2 -18826.754} C_VEL
LIN {X 0,Y 252.048,Z 367.177,A -85,B 0,C 180,E1 -18829.548,E2 -18829.548} C_VEL
LIN {X 0,Y 254.162,Z 357.941,A -85,B 0,C 180,E1 -18831.919,E2 -18831.919} C_VEL
LIN {X 0,Y 256.541,Z 347.741,A -85,B 0,C 180,E1 -18834.048,E2 -18834.048} C_VEL
LIN {X 0,Y 259.033,Z 335.909,A -85,B 0,C 180,E1 -18836.049,E2 -18836.049} C_VEL
LIN {X 0,Y 261.319,Z 324.115,A -85,B 0,C 180,E1 -18837.64,E2 -18837.64} C_VEL
LIN {X 0,Y 263.477,Z 311.157,A -85,B 0,C 180,E1 -18839.021,E2 -18839.021} C_VEL
LIN {X 0,Y 265.41,Z 297.796,A -85,B 0,C 180,E1 -18840.096,E2 -18840.096} C_VEL
LIN {X 0,Y 266.908,Z 284.153,A -85,B 0,C 180,E1 -18840.894,E2 -18840.894} C_VEL
LIN {X 0,Y 267.876,Z 270.372,A -85,B 0,C 180,E1 -18841.429,E2 -18841.429} C_VEL
LIN {X 0,Y 270.779,Z 190.093,A -85,B 0,C 180,E1 -18843.51,E2 -18843.51} C_VEL
LIN {X 0,Y 268.539,Z 174.764,A -85,B 0,C 180,E1 -18844.265,E2 -18844.265} C_VEL
LIN {X 0,Y 260.746,Z 155.661,A -85,B 0,C 180,E1 -18845.933,E2 -18845.933} C_VEL
LIN {X 0,Y 252.989,Z 139.613,A -85,B 0,C 180,E1 -18847.628,E2 -18847.628} C_VEL
LIN {X 0,Y 251.32,Z 136.029,A -85,B 0,C 180,E1 -18848.05,E2 -18848.05} C_VEL
LIN {X 0,Y 249.017,Z 127.593,A -85,B 0,C 180,E1 -18851.577,E2 -18851.577} C_VEL
LIN {X 0,Y 249.019,Z 127.591,A -85,B 0,C 180,E1 -18855.125,E2 -18855.125} C_VEL
LIN {X 0,Y 249.08,Z 127.581,A -85,B 0,C 180,E1 -18857.377,E2 -18857.377} C_VEL
LIN {X 0,Y 249.051,Z 127.565,A -85,B 0,C 180,E1 -18861.624,E2 -18861.624} C_VEL
LIN {X 0,Y 249.06,Z 127.582,A -85,B 0,C 180,E1 -18865.642,E2 -18865.642} C_VEL
LIN {X 0,Y 249.051,Z 127.585,A -85,B 0,C 180,E1 -18869.473,E2 -18869.473} C_VEL
LIN {X 0,Y 249.074,Z 127.586,A -85,B 0,C 180,E1 -18873.163,E2 -18873.163} C_VEL
LIN {X 0,Y 249.079,Z 127.577,A -85,B 0,C 180,E1 -18876.733,E2 -18876.733} C_VEL
LIN {X 0,Y 249.11,Z 127.576,A -85,B 0,C 180,E1 -18880.212,E2 -18880.212} C_VEL
LIN {X 0,Y 249.241,Z 127.562,A -85,B 0,C 180,E1 -18883.622,E2 -18883.622} C_VEL
LIN {X 0,Y 249.252,Z 127.553,A -85,B 0,C 180,E1 -18888.617,E2 -18888.617} C_VEL
LIN {X 0,Y 249.468,Z 127.534,A -85,B 0,C 180,E1 -18891.903,E2 -18891.903} C_VEL
LIN {X 0,Y 249.434,Z 127.54,A -85,B 0,C 180,E1 -18896.77,E2 -18896.77} C_VEL
LIN {X 0,Y 249.727,Z 127.497,A -85,B 0,C 180,E1 -18900,E2 -18900} C_VEL
LIN {X 0,Y 249.431,Z 127.529,A -85,B 0,C 180,E1 -18903.231,E2 -18903.231} C_VEL
LIN {X 0,Y 249.431,Z 127.538,A -85,B 0,C 180,E1 -18906.566,E2 -18906.566} C_VEL
LIN {X 0,Y 249.343,Z 127.535,A -85,B 0,C 180,E1 -18909.737,E2 -18909.737} C_VEL
LIN {X 0,Y 249.205,Z 127.566,A -85,B 0,C 180,E1 -18914.704,E2 -18914.704} C_VEL
LIN {X 0,Y 249.14,Z 127.562,A -85,B 0,C 180,E1 -18918.078,E2 -18918.078} C_VEL
LIN {X 0,Y 249.104,Z 127.582,A -85,B 0,C 180,E1 -18921.517,E2 -18921.517} C_VEL
LIN {X 0,Y 249.13,Z 127.564,A -85,B 0,C 180,E1 -18925.483,E2 -18925.483} C_VEL
LIN {X 0,Y 249.083,Z 127.584,A -85,B 0,C 180,E1 -18928.994,E2 -18928.994} C_VEL
LIN {X 0,Y 249.03,Z 127.582,A -85,B 0,C 180,E1 -18932.426,E2 -18932.426} C_VEL
LIN {X 0,Y 249.048,Z 127.582,A -85,B 0,C 180,E1 -18936.343,E2 -18936.343} C_VEL
LIN {X 0,Y 249.006,Z 127.593,A -85,B 0,C 180,E1 -18940.479,E2 -18940.479} C_VEL
LIN {X 0,Y 249.008,Z 127.59,A -85,B 0,C 180,E1 -18944.879,E2 -18944.879} C_VEL
LIN {X 0,Y 249.019,Z 127.591,A -85,B 0,C 180,E1 -18947.364,E2 -18947.364} C_VEL
LIN {X 0,Y 249.044,Z 127.572,A -85,B 0,C 180,E1 -18952.201,E2 -18952.201} C_VEL
LIN {X 0,Y 249.044,Z 127.587,A -85,B 0,C 180,E1 -18955.64,E2 -18955.64} C_VEL
LIN {X 0,Y 249.052,Z 127.781,A -85,B 0,C 180,E1 -18957.703,E2 -18957.703} C_VEL
LIN {X 0,Y 250.203,Z 130.729,A -85,B 0,C 180,E1 -18957.996,E2 -18957.996} C_VEL
LIN {X 0,Y 251.697,Z 132.875,A -85,B 0,C 180,E1 -18958.312,E2 -18958.312} C_VEL
LIN {X 0,Y 255.528,Z 139.637,A -85,B 0,C 180,E1 -18959.142,E2 -18959.142} C_VEL
LIN {X 0,Y 262.827,Z 154.569,A -85,B 0,C 180,E1 -18960.703,E2 -18960.703} C_VEL
LIN {X 0,Y 270.068,Z 172.054,A -85,B 0,C 180,E1 -18962.226,E2 -18962.226} C_VEL
LIN {X 0,Y 271.351,Z 175.687,A -85,B 0,C 180,E1 -18962.501,E2 -18962.501} C_VEL
LIN {X 0,Y 268.001,Z 263.436,A -85,B 0,C 180,E1 -18964.778,E2 -18964.778} C_VEL
LIN {X 0,Y 267.021,Z 277.263,A -85,B 0,C 180,E1 -18965.406,E2 -18965.406} C_VEL
LIN {X 0,Y 265.565,Z 290.819,A -85,B 0,C 180,E1 -18966.302,E2 -18966.302} C_VEL
LIN {X 0,Y 263.705,Z 304.012,A -85,B 0,C 180,E1 -18967.474,E2 -18967.474} C_VEL
LIN {X 0,Y 261.485,Z 316.733,A -85,B 0,C 180,E1 -18968.932,E2 -18968.932} C_VEL
LIN {X 0,Y 259.307,Z 328.282,A -85,B 0,C 180,E1 -18970.609,E2 -18970.609} C_VEL
LIN {X 0,Y 257.029,Z 338.879,A -85,B 0,C 180,E1 -18972.496,E2 -18972.496} C_VEL
LIN {X 0,Y 254.565,Z 349.389,A -85,B 0,C 180,E1 -18974.795,E2 -18974.795} C_VEL
LIN {X 0,Y 252.602,Z 358.057,A -85,B 0,C 180,E1 -18977.14,E2 -18977.14} C_VEL
LIN {X 0,Y 250.651,Z 366.384,A -85,B 0,C 180,E1 -18979.907,E2 -18979.907} C_VEL
LIN {X 0,Y 249.073,Z 373.093,A -85,B 0,C 180,E1 -18982.705,E2 -18982.705} C_VEL
LIN {X 0,Y 248.074,Z 377.706,A -85,B 0,C 180,E1 -18985.125,E2 -18985.125} C_VEL
LIN {X 0,Y 247.314,Z 382.497,A -85,B 0,C 180,E1 -18988.372,E2 -18988.372} C_VEL
LIN {X 0,Y 246.995,Z 385.817,A -85,B 0,C 180,E1 -18991.631,E2 -18991.631} C_VEL
LIN {X 0,Y 246.884,Z 387.758,A -85,B 0,C 180,E1 -18994.899,E2 -18994.899} C_VEL
LIN {X 0,Y 246.811,Z 388.369,A -85,B 0,C 180,E1 -18998.186,E2 -18998.186} C_VEL
LIN {X 0,Y 247.011,Z 387.649,A -85,B 0,C 180,E1 -19001.488,E2 -19001.488} C_VEL
LIN {X 0,Y 247.815,Z 385.574,A -85,B 0,C 180,E1 -19004.788,E2 -19004.788} C_VEL
LIN {X 0,Y 248.968,Z 382.089,A -85,B 0,C 180,E1 -19008.09,E2 -19008.09} C_VEL
LIN {X 0,Y 250.793,Z 377.078,A -85,B 0,C 180,E1 -19011.365,E2 -19011.365} C_VEL
LIN {X 0,Y 252.564,Z 372.2,A -85,B 0,C 180,E1 -19013.796,E2 -19013.796} C_VEL
LIN {X 0,Y 255.125,Z 365.139,A -85,B 0,C 180,E1 -19016.593,E2 -19016.593} C_VEL
LIN {X 0,Y 257.775,Z 357.73,A -85,B 0,C 180,E1 -19018.943,E2 -19018.943} C_VEL
LIN {X 0,Y 260.711,Z 348.788,A -85,B 0,C 180,E1 -19021.26,E2 -19021.26} C_VEL
LIN {X 0,Y 263.483,Z 339.891,A -85,B 0,C 180,E1 -19023.148,E2 -19023.148} C_VEL
LIN {X 0,Y 266.694,Z 329.257,A -85,B 0,C 180,E1 -19024.971,E2 -19024.971} C_VEL
LIN {X 0,Y 269.549,Z 317.757,A -85,B 0,C 180,E1 -19026.591,E2 -19026.591} C_VEL
LIN {X 0,Y 272.555,Z 304.813,A -85,B 0,C 180,E1 -19027.998,E2 -19027.998} C_VEL
LIN {X 0,Y 274.675,Z 292.632,A -85,B 0,C 180,E1 -19029.055,E2 -19029.055} C_VEL
LIN {X 0,Y 276.599,Z 278.449,A -85,B 0,C 180,E1 -19029.974,E2 -19029.974} C_VEL
LIN {X 0,Y 277.989,Z 264.269,A -85,B 0,C 180,E1 -19030.587,E2 -19030.587} C_VEL
LIN {X 0,Y 281.725,Z 186.538,A -85,B 0,C 180,E1 -19032.529,E2 -19032.529} C_VEL
LIN {X 0,Y 280.717,Z 183.564,A -85,B 0,C 180,E1 -19032.794,E2 -19032.794} C_VEL
LIN {X 0,Y 274.898,Z 171.199,A -85,B 0,C 180,E1 -19034.222,E2 -19034.222} C_VEL
LIN {X 0,Y 267.817,Z 157.758,A -85,B 0,C 180,E1 -19036.033,E2 -19036.033} C_VEL
LIN {X 0,Y 260.852,Z 145.975,A -85,B 0,C 180,E1 -19037.915,E2 -19037.915} C_VEL
LIN {X 0,Y 254.815,Z 136.676,A -85,B 0,C 180,E1 -19039.648,E2 -19039.648} C_VEL
LIN {X 0,Y 252.613,Z 133.521,A -85,B 0,C 180,E1 -19040.306,E2 -19040.306} C_VEL
LIN {X 0,Y 251.92,Z 132.481,A -85,B 0,C 180,E1 -19040.519,E2 -19040.519} C_VEL
LIN {X 0,Y 249.87,Z 130.215,A -85,B 0,C 180,E1 -19041.128,E2 -19041.128} C_VEL
LIN {X 0,Y 249.033,Z 127.819,A -85,B 0,C 180,E1 -19041.491,E2 -19041.491} C_VEL
LIN {X 0,Y 249.022,Z 127.586,A -85,B 0,C 180,E1 -19042.207,E2 -19042.207} C_VEL
LIN {X 0,Y 249.044,Z 127.589,A -85,B 0,C 180,E1 -19045.639,E2 -19045.639} C_VEL
LIN {X 0,Y 249.004,Z 127.587,A -85,B 0,C 180,E1 -19049.466,E2 -19049.466} C_VEL
LIN {X 0,Y 249.037,Z 127.58,A -85,B 0,C 180,E1 -19053.158,E2 -19053.158} C_VEL
LIN {X 0,Y 249.055,Z 127.579,A -85,B 0,C 180,E1 -19056.73,E2 -19056.73} C_VEL
LIN {X 0,Y 249.092,Z 127.581,A -85,B 0,C 180,E1 -19060.21,E2 -19060.21} C_VEL
LIN {X 0,Y 249.197,Z 127.569,A -85,B 0,C 180,E1 -19063.619,E2 -19063.619} C_VEL
LIN {X 0,Y 249.244,Z 127.565,A -85,B 0,C 180,E1 -19068.616,E2 -19068.616} C_VEL
LIN {X 0,Y 249.32,Z 127.542,A -85,B 0,C 180,E1 -19070.052,E2 -19070.052} C_VEL
LIN {X 0,Y 248.736,Z 127.618,A -85,B 0,C 180,E1 -19071.399,E2 -19071.399} C_VEL
LIN {X 0,Y 245.853,Z 127.986,A -85,B 0,C 180,E1 -19073.596,E2 -19073.596} C_VEL
LIN {X 0,Y 243.412,Z 128.28,A -85,B 0,C 180,E1 -19075.386,E2 -19075.386} C_VEL
LIN {X 0,Y 242.458,Z 128.394,A -85,B 0,C 180,E1 -19076.776,E2 -19076.776} C_VEL
LIN {X 0,Y 242.434,Z 128.399,A -85,B 0,C 180,E1 -19077.247,E2 -19077.247} C_VEL
LIN {X 0,Y 242.686,Z 128.371,A -85,B 0,C 180,E1 -19080,E2 -19080} C_VEL
LIN {X 0,Y 242.634,Z 128.371,A -85,B 0,C 180,E1 -19081.66,E2 -19081.66} C_VEL
LIN {X 0,Y 242.404,Z 128.399,A -85,B 0,C 180,E1 -19086.659,E2 -19086.659} C_VEL
LIN {X 0,Y 242.269,Z 128.426,A -85,B 0,C 180,E1 -19090.023,E2 -19090.023} C_VEL
LIN {X 0,Y 242.168,Z 128.434,A -85,B 0,C 180,E1 -19095.14,E2 -19095.14} C_VEL
LIN {X 0,Y 242.075,Z 128.454,A -85,B 0,C 180,E1 -19098.624,E2 -19098.624} C_VEL
LIN {X 0,Y 242.014,Z 128.457,A -85,B 0,C 180,E1 -19102.18,E2 -19102.18} C_VEL
LIN {X 0,Y 242.068,Z 128.446,A -85,B 0,C 180,E1 -19105.838,E2 -19105.838} C_VEL
LIN {X 0,Y 242.008,Z 128.456,A -85,B 0,C 180,E1 -19109.583,E2 -19109.583} C_VEL
LIN {X 0,Y 241.989,Z 128.464,A -85,B 0,C 180,E1 -19113.491,E2 -19113.491} C_VEL
LIN {X 0,Y 241.991,Z 128.461,A -85,B 0,C 180,E1 -19117.581,E2 -19117.581} C_VEL
LIN {X 0,Y 241.952,Z 128.548,A -85,B 0,C 180,E1 -19119.531,E2 -19119.531} C_VEL
LIN {X 0,Y 244.124,Z 135.399,A -85,B 0,C 180,E1 -19123.31,E2 -19123.31} C_VEL
LIN {X 0,Y 247.126,Z 139.982,A -85,B 0,C 180,E1 -19124.309,E2 -19124.309} C_VEL
LIN {X 0,Y 252.428,Z 148.452,A -85,B 0,C 180,E1 -19125.986,E2 -19125.986} C_VEL
LIN {X 0,Y 257.043,Z 156.008,A -85,B 0,C 180,E1 -19127.357,E2 -19127.357} C_VEL
LIN {X 0,Y 264.709,Z 170.142,A -85,B 0,C 180,E1 -19129.521,E2 -19129.521} C_VEL
LIN {X 0,Y 271.749,Z 184.913,A -85,B 0,C 180,E1 -19131.4,E2 -19131.4} C_VEL
LIN {X 0,Y 275.456,Z 193.872,A -85,B 0,C 180,E1 -19132.37,E2 -19132.37} C_VEL
LIN {X 0,Y 275.735,Z 197.598,A -85,B 0,C 180,E1 -19132.543,E2 -19132.543} C_VEL
LIN {X 0,Y 272,Z 274.448,A -85,B 0,C 180,E1 -19134.51,E2 -19134.51} C_VEL
LIN {X 0,Y 270.432,Z 288.845,A -85,B 0,C 180,E1 -19135.128,E2 -19135.128} C_VEL
LIN {X 0,Y 268.364,Z 302.12,A -85,B 0,C 180,E1 -19135.96,E2 -19135.96} C_VEL
LIN {X 0,Y 265.947,Z 314.261,A -85,B 0,C 180,E1 -19136.972,E2 -19136.972} C_VEL
LIN {X 0,Y 262.938,Z 327.038,A -85,B 0,C 180,E1 -19138.362,E2 -19138.362} C_VEL
LIN {X 0,Y 259.768,Z 339.007,A -85,B 0,C 180,E1 -19140.032,E2 -19140.032} C_VEL
LIN {X 0,Y 256.634,Z 349.323,A -85,B 0,C 180,E1 -19141.81,E2 -19141.81} C_VEL
LIN {X 0,Y 253.08,Z 359.901,A -85,B 0,C 180,E1 -19144.063,E2 -19144.063} C_VEL
LIN {X 0,Y 250.011,Z 368.647,A -85,B 0,C 180,E1 -19146.385,E2 -19146.385} C_VEL
LIN {X 0,Y 246.886,Z 377.053,A -85,B 0,C 180,E1 -19149.155,E2 -19149.155} C_VEL
LIN {X 0,Y 244.731,Z 382.932,A -85,B 0,C 180,E1 -19151.585,E2 -19151.585} C_VEL
LIN {X 0,Y 242.57,Z 389.234,A -85,B 0,C 180,E1 -19154.885,E2 -19154.885} C_VEL
LIN {X 0,Y 241.004,Z 393.917,A -85,B 0,C 180,E1 -19158.221,E2 -19158.221} C_VEL
LIN {X 0,Y 240.142,Z 397.123,A -85,B 0,C 180,E1 -19161.585,E2 -19161.585} C_VEL
LIN {X 0,Y 239.766,Z 398.966,A -85,B 0,C 180,E1 -19164.955,E2 -19164.955} C_VEL
LIN {X 0,Y 239.799,Z 399.485,A -85,B 0,C 180,E1 -19168.32,E2 -19168.32} C_VEL
LIN {X 0,Y 239.843,Z 399.245,A -85,B 0,C 180,E1 -19170,E2 -19170} C_VEL
LIN {X 0,Y 239.806,Z 398.667,A -85,B 0,C 180,E1 -19171.679,E2 -19171.679} C_VEL
LIN {X 0,Y 239.766,Z 396.486,A -85,B 0,C 180,E1 -19175.045,E2 -19175.045} C_VEL
LIN {X 0,Y 240.067,Z 392.886,A -85,B 0,C 180,E1 -19178.417,E2 -19178.417} C_VEL
LIN {X 0,Y 240.755,Z 387.755,A -85,B 0,C 180,E1 -19181.791,E2 -19181.791} C_VEL
LIN {X 0,Y 241.772,Z 382.783,A -85,B 0,C 180,E1 -19184.305,E2 -19184.305} C_VEL
LIN {X 0,Y 243.083,Z 376.76,A -85,B 0,C 180,E1 -19186.805,E2 -19186.805} C_VEL
LIN {X 0,Y 244.61,Z 369.498,A -85,B 0,C 180,E1 -19189.293,E2 -19189.293} C_VEL
LIN {X 0,Y 246.737,Z 360.764,A -85,B 0,C 180,E1 -19191.733,E2 -19191.733} C_VEL
LIN {X 0,Y 249.293,Z 350.171,A -85,B 0,C 180,E1 -19194.128,E2 -19194.128} C_VEL
LIN {X 0,Y 251.772,Z 339.489,A -85,B 0,C 180,E1 -19196.081,E2 -19196.081} C_VEL
LIN {X 0,Y 254.124,Z 327.881,A -85,B 0,C 180,E1 -19197.81,E2 -19197.81} C_VEL
LIN {X 0,Y 256.493,Z 314.985,A -85,B 0,C 180,E1 -19199.326,E2 -19199.326} C_VEL
LIN {X 0,Y 258.587,Z 301.671,A -85,B 0,C 180,E1 -19200.524,E2 -19200.524} C_VEL
LIN {X 0,Y 260.342,Z 287.188,A -85,B 0,C 180,E1 -19201.479,E2 -19201.479} C_VEL
LIN {X 0,Y 261.54,Z 272.502,A -85,B 0,C 180,E1 -19202.11,E2 -19202.11} C_VEL
LIN {X 0,Y 264.699,Z 191.219,A -85,B 0,C 180,E1 -19204.26,E2 -19204.26} C_VEL
LIN {X 0,Y 262.822,Z 177.662,A -85,B 0,C 180,E1 -19204.939,E2 -19204.939} C_VEL
LIN {X 0,Y 255.838,Z 160.329,A -85,B 0,C 180,E1 -19206.498,E2 -19206.498} C_VEL
LIN {X 0,Y 248.269,Z 144.194,A -85,B 0,C 180,E1 -19208.229,E2 -19208.229} C_VEL
LIN {X 0,Y 243.971,Z 135.827,A -85,B 0,C 180,E1 -19209.288,E2 -19209.288} C_VEL
LIN {X 0,Y 241.983,Z 128.469,A -85,B 0,C 180,E1 -19212.468,E2 -19212.468} C_VEL
LIN {X 0,Y 242.001,Z 128.462,A -85,B 0,C 180,E1 -19216.554,E2 -19216.554} C_VEL
LIN {X 0,Y 242.009,Z 128.445,A -85,B 0,C 180,E1 -19220.292,E2 -19220.292} C_VEL
LIN {X 0,Y 242.036,Z 128.46,A -85,B 0,C 180,E1 -19224.498,E2 -19224.498} C_VEL
LIN {X 0,Y 241.975,Z 128.468,A -85,B 0,C 180,E1 -19228.48,E2 -19228.48} C_VEL
LIN {X 0,Y 242.008,Z 128.462,A -85,B 0,C 180,E1 -19232.313,E2 -19232.313} C_VEL
LIN {X 0,Y 242.057,Z 128.449,A -85,B 0,C 180,E1 -19236.016,E2 -19236.016} C_VEL
LIN {X 0,Y 242.037,Z 128.457,A -85,B 0,C 180,E1 -19239.608,E2 -19239.608} C_VEL
LIN {X 0,Y 242.162,Z 128.445,A -85,B 0,C 180,E1 -19243.278,E2 -19243.278} C_VEL
LIN {X 0,Y 242.186,Z 128.43,A -85,B 0,C 180,E1 -19248.28,E2 -19248.28} C_VEL
LIN {X 0,Y 242.416,Z 128.412,A -85,B 0,C 180,E1 -19251.665,E2 -19251.665} C_VEL
LIN {X 0,Y 242.256,Z 128.422,A -85,B 0,C 180,E1 -19255.007,E2 -19255.007} C_VEL
LIN {X 0,Y 242.635,Z 128.387,A -85,B 0,C 180,E1 -19258.34,E2 -19258.34} C_VEL
LIN {X 0,Y 242.635,Z 128.369,A -85,B 0,C 180,E1 -19261.66,E2 -19261.66} C_VEL
LIN {X 0,Y 242.408,Z 128.413,A -85,B 0,C 180,E1 -19266.66,E2 -19266.66} C_VEL
LIN {X 0,Y 242.267,Z 128.415,A -85,B 0,C 180,E1 -19270.024,E2 -19270.024} C_VEL
LIN {X 0,Y 242.167,Z 128.443,A -85,B 0,C 180,E1 -19275.141,E2 -19275.141} C_VEL
LIN {X 0,Y 242.079,Z 128.443,A -85,B 0,C 180,E1 -19278.624,E2 -19278.624} C_VEL
LIN {X 0,Y 242.05,Z 128.457,A -85,B 0,C 180,E1 -19282.177,E2 -19282.177} C_VEL
LIN {X 0,Y 242.067,Z 128.445,A -85,B 0,C 180,E1 -19285.839,E2 -19285.839} C_VEL
LIN {X 0,Y 242.03,Z 128.458,A -85,B 0,C 180,E1 -19289.581,E2 -19289.581} C_VEL
LIN {X 0,Y 241.981,Z 128.467,A -85,B 0,C 180,E1 -19293.493,E2 -19293.493} C_VEL
LIN {X 0,Y 241.989,Z 128.459,A -85,B 0,C 180,E1 -19297.582,E2 -19297.582} C_VEL
LIN {X 0,Y 241.939,Z 128.464,A -85,B 0,C 180,E1 -19301.923,E2 -19301.923} C_VEL
LIN {X 0,Y 241.938,Z 128.467,A -85,B 0,C 180,E1 -19306.571,E2 -19306.571} C_VEL
LIN {X 0,Y 241.957,Z 128.451,A -85,B 0,C 180,E1 -19310.282,E2 -19310.282} C_VEL
LIN {X 0,Y 241.989,Z 128.468,A -85,B 0,C 180,E1 -19314.49,E2 -19314.49} C_VEL
LIN {X 0,Y 241.981,Z 128.472,A -85,B 0,C 180,E1 -19316.508,E2 -19316.508} C_VEL
LIN {X 0,Y 242.922,Z 131.255,A -85,B 0,C 180,E1 -19316.779,E2 -19316.779} C_VEL
LIN {X 0,Y 244.629,Z 133.711,A -85,B 0,C 180,E1 -19317.165,E2 -19317.165} C_VEL
LIN {X 0,Y 250.263,Z 143.241,A -85,B 0,C 180,E1 -19318.437,E2 -19318.437} C_VEL
LIN {X 0,Y 257.83,Z 158.962,A -85,B 0,C 180,E1 -19320.127,E2 -19320.127} C_VEL
LIN {X 0,Y 264.668,Z 175.772,A -85,B 0,C 180,E1 -19321.628,E2 -19321.628} C_VEL
LIN {X 0,Y 265.221,Z 177.63,A -85,B 0,C 180,E1 -19321.761,E2 -19321.761} C_VEL
LIN {X 0,Y 261.82,Z 263.495,A -85,B 0,C 180,E1 -19324.032,E2 -19324.032} C_VEL
LIN {X 0,Y 260.795,Z 277.367,A -85,B 0,C 180,E1 -19324.672,E2 -19324.672} C_VEL
LIN {X 0,Y 259.279,Z 290.94,A -85,B 0,C 180,E1 -19325.584,E2 -19325.584} C_VEL
LIN {X 0,Y 257.509,Z 303.265,A -85,B 0,C 180,E1 -19326.688,E2 -19326.688} C_VEL
LIN {X 0,Y 255.168,Z 316.167,A -85,B 0,C 180,E1 -19328.172,E2 -19328.172} C_VEL
LIN {X 0,Y 252.908,Z 327.845,A -85,B 0,C 180,E1 -19329.887,E2 -19329.887} C_VEL
